KUKA KRL program: MyProgram_012().src

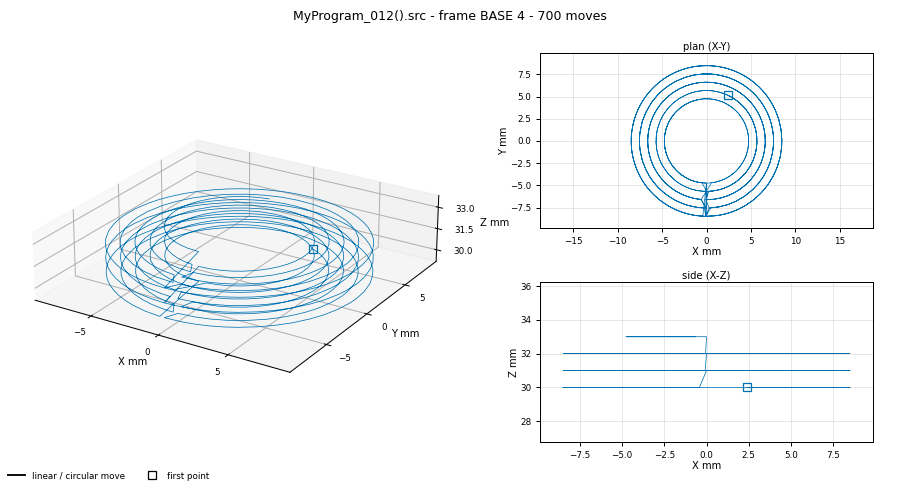
[picture p0: tool path of MyProgram_012().src in frame BASE 4, 700 of 700 moves have a stored position in this frame; points joined in program order, loops and branches not executed]
&ACCESS RVP
&REL 1
&PARAM TEMPLATE = C:\KRC\Roboter\Template\vorgabe
&PARAM EDITMASK = *
DEF MyProgram_012()
; ---- Setting reference (Base) ----
$BASE = BASE_DATA[4]

; --------------------------
; ---- Setting tool (TCP) ----
$TOOL = TOOL_DATA[3]
; --------------------------

$VEL.CP = VEL_APROX_PRINT
Startdeposition()
$VEL.CP = VEL_PRINT
LIN {X 2.4123,Y 5.1442,Z 30,A -2.4126,B 0,C 0,E1 0.1598,E2 90.0723} C_DIS
LIN {X 3.1461,Y 4.7312,Z 30,A -2.403,B 0,C 0,E1 0.1598,E2 90.0723} C_DIS
LIN {X 3.8114,Y 4.215,Z 30,A -2.4004,B 0,C 0,E1 0.1598,E2 90.0723} C_DIS
LIN {X 4.392,Y 3.6051,Z 30,A -2.4048,B 0,C 0,E1 0.1598,E2 90.0721} C_DIS
LIN {X 4.8767,Y 2.9165,Z 30,A -2.4161,B 0,C 0,E1 0.1598,E2 90.0721} C_DIS
LIN {X 5.2536,Y 2.1636,Z 30,A -2.4342,B 0,C 0,E1 0.1598,E2 90.072} C_DIS
LIN {X 5.5158,Y 1.3634,Z 30,A -2.4585,B 0,C 0,E1 0.1598,E2 90.072} C_DIS
LIN {X 5.6573,Y 0.5334,Z 30,A -2.4886,B 0,C 0,E1 0.1598,E2 90.0719} C_DIS
LIN {X 5.6741,Y -0.3085,Z 30,A -2.5238,B 0,C 0,E1 0.1598,E2 90.0719} C_DIS
LIN {X 5.567,Y -1.1438,Z 30,A -2.5633,B 0,C 0,E1 0.1598,E2 90.0718} C_DIS
LIN {X 5.3364,Y -1.9538,Z 30,A -2.6062,B 0,C 0,E1 0.1598,E2 90.0718} C_DIS
LIN {X 4.9891,Y -2.721,Z 30,A -2.6517,B 0,C 0,E1 0.1598,E2 90.0718} C_DIS
LIN {X 4.5312,Y -3.4277,Z 30,A -2.6986,B 0,C 0,E1 0.1598,E2 90.0718} C_DIS
LIN {X 3.9758,Y -4.0606,Z 30,A -2.746,B 0,C 0,E1 0.1598,E2 90.0718} C_DIS
LIN {X 3.3312,Y -4.6025,Z 30,A -2.7928,B 0,C 0,E1 0.1598,E2 90.0718} C_DIS
LIN {X 2.6147,Y -5.0448,Z 30,A -2.8379,B 0,C 0,E1 0.1598,E2 90.0717} C_DIS
LIN {X 1.8405,Y -5.3759,Z 30,A -2.8805,B 0,C 0,E1 0.1598,E2 90.0717} C_DIS
LIN {X 1.0258,Y -5.5886,Z 30,A -2.9194,B 0,C 0,E1 0.1598,E2 90.0717} C_DIS
LIN {X 0.1887,Y -5.6795,Z 30,A -2.954,B 0,C 0,E1 0.1598,E2 90.0717} C_DIS
LIN {X 0.1887,Y -5.6795,Z 30,A -2.954,B 0,C 0,E1 0.1598,E2 90.0717} C_DIS
Enddeposition()
LIN {X -0.0561,Y -6.623,Z 30,A -3.0021,B 0,C 0,E1 0.1598,E2 90.0704} C_DIS
Startdeposition()
$VEL.CP = VEL_PRINT
LIN {X 0.9035,Y -6.5557,Z 30,A -2.9651,B 0,C 0,E1 0.1598,E2 90.0716} C_DIS
LIN {X 1.6588,Y -6.4076,Z 30,A -2.9312,B 0,C 0,E1 0.1598,E2 90.0716} C_DIS
LIN {X 2.3917,Y -6.1725,Z 30,A -2.8943,B 0,C 0,E1 0.1598,E2 90.0716} C_DIS
LIN {X 3.0924,Y -5.8533,Z 30,A -2.855,B 0,C 0,E1 0.1598,E2 90.0717} C_DIS
LIN {X 3.7497,Y -5.4527,Z 30,A -2.8138,B 0,C 0,E1 0.1598,E2 90.0717} C_DIS
LIN {X 4.3594,Y -4.983,Z 30,A -2.7714,B 0,C 0,E1 0.1598,E2 90.0717} C_DIS
LIN {X 4.9078,Y -4.4428,Z 30,A -2.7282,B 0,C 0,E1 0.1598,E2 90.0717} C_DIS
LIN {X 5.3882,Y -3.8416,Z 30,A -2.6849,B 0,C 0,E1 0.1598,E2 90.0718} C_DIS
LIN {X 5.7983,Y -3.1903,Z 30,A -2.6421,B 0,C 0,E1 0.1598,E2 90.0718} C_DIS
LIN {X 6.1306,Y -2.4959,Z 30,A -2.6003,B 0,C 0,E1 0.1598,E2 90.0718} C_DIS
LIN {X 6.3796,Y -1.7675,Z 30,A -2.5601,B 0,C 0,E1 0.1598,E2 90.0718} C_DIS
LIN {X 6.5402,Y -1.0147,Z 30,A -2.5221,B 0,C 0,E1 0.1598,E2 90.0718} C_DIS
LIN {X 6.613,Y -0.2485,Z 30,A -2.4868,B 0,C 0,E1 0.1598,E2 90.0719} C_DIS
LIN {X 6.5976,Y 0.5209,Z 30,A -2.4546,B 0,C 0,E1 0.1598,E2 90.0719} C_DIS
LIN {X 6.4945,Y 1.2838,Z 30,A -2.4259,B 0,C 0,E1 0.1598,E2 90.072} C_DIS
LIN {X 6.2995,Y 2.0284,Z 30,A -2.4014,B 0,C 0,E1 0.1598,E2 90.072} C_DIS
LIN {X 6.0209,Y 2.7458,Z 30,A -2.3812,B 0,C 0,E1 0.1598,E2 90.072} C_DIS
LIN {X 5.6618,Y 3.4265,Z 30,A -2.3655,B 0,C 0,E1 0.1598,E2 90.0721} C_DIS
LIN {X 5.2259,Y 4.0609,Z 30,A -2.3547,B 0,C 0,E1 0.1598,E2 90.0721} C_DIS
LIN {X 4.7191,Y 4.6402,Z 30,A -2.3488,B 0,C 0,E1 0.1598,E2 90.0722} C_DIS
LIN {X 4.1479,Y 5.156,Z 30,A -2.348,B 0,C 0,E1 0.1598,E2 90.0722} C_DIS
LIN {X 3.5214,Y 5.6029,Z 30,A -2.3521,B 0,C 0,E1 0.1598,E2 90.0723} C_DIS
LIN {X 2.8468,Y 5.9734,Z 30,A -2.3613,B 0,C 0,E1 0.1598,E2 90.0723} C_DIS
LIN {X 2.1347,Y 6.2654,Z 30,A -2.3753,B 0,C 0,E1 0.1598,E2 90.0723} C_DIS
LIN {X 1.393,Y 6.4721,Z 30,A -2.3939,B 0,C 0,E1 0.1598,E2 90.0723} C_DIS
LIN {X 0.6321,Y 6.5887,Z 30,A -2.417,B 0,C 0,E1 0.1598,E2 90.0723} C_DIS
LIN {X -0.137,Y 6.616,Z 30,A -2.4443,B 0,C 0,E1 0.1598,E2 90.0723} C_DIS
LIN {X -0.9042,Y 6.5562,Z 30,A -2.4751,B 0,C 0,E1 0.1598,E2 90.0723} C_DIS
LIN {X -1.6593,Y 6.4071,Z 30,A -2.5093,B 0,C 0,E1 0.1598,E2 90.0723} C_DIS
LIN {X -2.3924,Y 6.1721,Z 30,A -2.5462,B 0,C 0,E1 0.1598,E2 90.0722} C_DIS
LIN {X -3.093,Y 5.8529,Z 30,A -2.5855,B 0,C 0,E1 0.1598,E2 90.0721} C_DIS
LIN {X -3.7524,Y 5.4556,Z 30,A -2.6266,B 0,C 0,E1 0.1598,E2 90.072} C_DIS
LIN {X -4.3593,Y 4.9822,Z 30,A -2.669,B 0,C 0,E1 0.1598,E2 90.072} C_DIS
LIN {X -4.9079,Y 4.4421,Z 30,A -2.712,B 0,C 0,E1 0.1598,E2 90.0718} C_DIS
LIN {X -5.3904,Y 3.8421,Z 30,A -2.7551,B 0,C 0,E1 0.1598,E2 90.0718} C_DIS
LIN {X -5.8017,Y 3.1913,Z 30,A -2.7977,B 0,C 0,E1 0.1598,E2 90.0716} C_DIS
LIN {X -6.132,Y 2.496,Z 30,A -2.8392,B 0,C 0,E1 0.1598,E2 90.0716} C_DIS
LIN {X -6.3803,Y 1.7674,Z 30,A -2.8791,B 0,C 0,E1 0.1598,E2 90.0715} C_DIS
LIN {X -6.5428,Y 1.015,Z 30,A -2.9168,B 0,C 0,E1 0.1598,E2 90.0714} C_DIS
LIN {X -6.6157,Y 0.2486,Z 30,A -2.9518,B 0,C 0,E1 0.1598,E2 90.0714} C_DIS
LIN {X -6.5995,Y -0.521,Z 30,A -2.9837,B 0,C 0,E1 0.1598,E2 90.0713} C_DIS
LIN {X -6.493,Y -1.2834,Z 30,A -3.0121,B 0,C 0,E1 0.1598,E2 90.0713} C_DIS
LIN {X -6.2988,Y -2.0281,Z 30,A -3.0364,B 0,C 0,E1 0.1598,E2 90.0713} C_DIS
LIN {X -6.0221,Y -2.7462,Z 30,A -3.0566,B 0,C 0,E1 0.1598,E2 90.0713} C_DIS
LIN {X -5.6621,Y -3.4265,Z 30,A -3.0722,B 0,C 0,E1 0.1598,E2 90.0713} C_DIS
LIN {X -5.2258,Y -4.0606,Z 30,A -3.083,B 0,C 0,E1 0.1598,E2 90.0713} C_DIS
LIN {X -4.7193,Y -4.6402,Z 30,A -3.089,B 0,C 0,E1 0.1598,E2 90.0713} C_DIS
LIN {X -4.1488,Y -5.157,Z 30,A -3.09,B 0,C 0,E1 0.1598,E2 90.0713} C_DIS
LIN {X -3.5234,Y -5.6058,Z 30,A -3.0861,B 0,C 0,E1 0.1598,E2 90.0713} C_DIS
LIN {X -2.8478,Y -5.9745,Z 30,A -3.077,B 0,C 0,E1 0.1598,E2 90.0713} C_DIS
LIN {X -2.1347,Y -6.2644,Z 30,A -3.0631,B 0,C 0,E1 0.1598,E2 90.0714} C_DIS
LIN {X -1.3938,Y -6.4732,Z 30,A -3.0448,B 0,C 0,E1 0.1598,E2 90.0714} C_DIS
LIN {X -0.6329,Y -6.5897,Z 30,A -3.0219,B 0,C 0,E1 0.1598,E2 90.0715} C_DIS
LIN {X -0.6329,Y -6.5897,Z 30,A -3.0219,B 0,C 0,E1 0.1598,E2 90.0715} C_DIS
Enddeposition()
LIN {X -0.0547,Y -7.5529,Z 30,A -3.0406,B 0,C 0,E1 0.1598,E2 90.0703} C_DIS
Startdeposition()
$VEL.CP = VEL_PRINT
LIN {X -0.7724,Y -7.5177,Z 30,A -3.0665,B 0,C 0,E1 0.1598,E2 90.0714} C_DIS
LIN {X -1.851,Y -7.322,Z 30,A -3.0978,B 0,C 0,E1 0.1598,E2 90.0714} C_DIS
LIN {X -2.6875,Y -7.0585,Z 30,A -3.1173,B 0,C 0,E1 0.1598,E2 90.0714} C_DIS
LIN {X -3.4877,Y -6.6995,Z 30,A -3.1314,B 0,C 0,E1 0.1598,E2 90.0714} C_DIS
LIN {X -4.5316,Y -6.0476,Z 30,A -3.1419,B 0,C 0,E1 0.1598,E2 90.0712} C_DIS
LIN {X -5.2966,Y -5.385,Z 30,A -3.1419,B 0,C 0,E1 0.1598,E2 90.0712} C_DIS
LIN {X -5.8428,Y -4.7872,Z 30,A -3.1367,B 0,C 0,E1 0.1598,E2 90.0712} C_DIS
LIN {X -6.3205,Y -4.1335,Z 30,A -3.1265,B 0,C 0,E1 0.1598,E2 90.0712} C_DIS
LIN {X -6.8204,Y -3.2535,Z 30,A -3.1074,B 0,C 0,E1 0.1598,E2 90.0709} C_DIS
LIN {X -7.2077,Y -2.2699,Z 30,A -3.08,B 0,C 0,E1 0.1598,E2 90.0709} C_DIS
LIN {X -7.497,Y -0.9548,Z 30,A -3.0348,B 0,C 0,E1 0.1598,E2 90.0707} C_DIS
LIN {X -7.5586,Y 0,Z 30,A -2.997,B 0,C 0,E1 0.1598,E2 90.071} C_DIS
LIN {X -7.4963,Y 0.9605,Z 30,A -2.9542,B 0,C 0,E1 0.1598,E2 90.0712} C_DIS
LIN {X -7.2248,Y 2.2151,Z 30,A -2.8909,B 0,C 0,E1 0.1598,E2 90.0709} C_DIS
LIN {X -6.777,Y 3.3346,Z 30,A -2.8272,B 0,C 0,E1 0.1598,E2 90.0711} C_DIS
LIN {X -6.1243,Y 4.4288,Z 30,A -2.7571,B 0,C 0,E1 0.1598,E2 90.0713} C_DIS
LIN {X -5.5112,Y 5.165,Z 30,A -2.7037,B 0,C 0,E1 0.1598,E2 90.0717} C_DIS
LIN {X -4.9608,Y 5.6982,Z 30,A -2.661,B 0,C 0,E1 0.1598,E2 90.0719} C_DIS
LIN {X -4.3575,Y 6.171,Z 30,A -2.6188,B 0,C 0,E1 0.1598,E2 90.0719} C_DIS
LIN {X -3.5431,Y 6.6752,Z 30,A -2.5675,B 0,C 0,E1 0.1598,E2 90.072} C_DIS
LIN {X -2.4286,Y 7.1518,Z 30,A -2.5062,B 0,C 0,E1 0.1598,E2 90.0721} C_DIS
LIN {X -1.5729,Y 7.3873,Z 30,A -2.4648,B 0,C 0,E1 0.1598,E2 90.0723} C_DIS
LIN {X -0.3721,Y 7.549,Z 30,A -2.4136,B 0,C 0,E1 0.1598,E2 90.0723} C_DIS
LIN {X 0.6118,Y 7.5328,Z 30,A -2.378,B 0,C 0,E1 0.1598,E2 90.0723} C_DIS
LIN {X 1.7598,Y 7.3459,Z 30,A -2.3435,B 0,C 0,E1 0.1598,E2 90.0724} C_DIS
LIN {X 2.486,Y 7.1371,Z 30,A -2.3255,B 0,C 0,E1 0.1598,E2 90.0724} C_DIS
LIN {X 3.3884,Y 6.7498,Z 30,A -2.3086,B 0,C 0,E1 0.1598,E2 90.0724} C_DIS
LIN {X 4.071,Y 6.3612,Z 30,A -2.2999,B 0,C 0,E1 0.1598,E2 90.0724} C_DIS
LIN {X 4.7103,Y 5.9047,Z 30,A -2.2957,B 0,C 0,E1 0.1598,E2 90.0724} C_DIS
LIN {X 5.2981,Y 5.3837,Z 30,A -2.2961,B 0,C 0,E1 0.1598,E2 90.0724} C_DIS
LIN {X 5.8284,Y 4.8041,Z 30,A -2.3011,B 0,C 0,E1 0.1598,E2 90.0723} C_DIS
LIN {X 6.2957,Y 4.1726,Z 30,A -2.3107,B 0,C 0,E1 0.1598,E2 90.0723} C_DIS
LIN {X 6.6959,Y 3.4965,Z 30,A -2.3247,B 0,C 0,E1 0.1598,E2 90.0722} C_DIS
LIN {X 7.0228,Y 2.7821,Z 30,A -2.343,B 0,C 0,E1 0.1598,E2 90.0722} C_DIS
LIN {X 7.3273,Y 1.8485,Z 30,A -2.3712,B 0,C 0,E1 0.1598,E2 90.0718} C_DIS
LIN {X 7.5275,Y 0.6253,Z 30,A -2.4155,B 0,C 0,E1 0.1598,E2 90.0714} C_DIS
LIN {X 7.556,Y -0.1257,Z 30,A -2.4469,B 0,C 0,E1 0.1598,E2 90.0718} C_DIS
LIN {X 7.4453,Y -1.2667,Z 30,A -2.4994,B 0,C 0,E1 0.1598,E2 90.0716} C_DIS
LIN {X 7.1403,Y -2.4763,Z 30,A -2.5621,B 0,C 0,E1 0.1598,E2 90.0714} C_DIS
LIN {X 6.7973,Y -3.3011,Z 30,A -2.6101,B 0,C 0,E1 0.1598,E2 90.0716} C_DIS
LIN {X 6.3336,Y -4.1158,Z 30,A -2.6619,B 0,C 0,E1 0.1598,E2 90.0716} C_DIS
LIN {X 5.8945,Y -4.7239,Z 30,A -2.7041,B 0,C 0,E1 0.1598,E2 90.0718} C_DIS
LIN {X 5.2662,Y -5.4196,Z 30,A -2.7567,B 0,C 0,E1 0.1598,E2 90.0716} C_DIS
LIN {X 4.2992,Y -6.2142,Z 30,A -2.826,B 0,C 0,E1 0.1598,E2 90.0716} C_DIS
LIN {X 3.3206,Y -6.7878,Z 30,A -2.8864,B 0,C 0,E1 0.1598,E2 90.0716} C_DIS
LIN {X 2.3699,Y -7.1764,Z 30,A -2.9379,B 0,C 0,E1 0.1598,E2 90.0716} C_DIS
LIN {X 1.4049,Y -7.4218,Z 30,A -2.9838,B 0,C 0,E1 0.1598,E2 90.0716} C_DIS
LIN {X 0.2911,Y -7.5523,Z 30,A -3.0302,B 0,C 0,E1 0.1598,E2 90.0716} C_DIS
LIN {X 0.2911,Y -7.5523,Z 30,A -3.0302,B 0,C 0,E1 0.1598,E2 90.0716} C_DIS
Enddeposition()
LIN {X -0.0783,Y -8.4901,Z 30,A -3.0826,B 0,C 0,E1 0.1598,E2 90.0703} C_DIS
Startdeposition()
$VEL.CP = VEL_PRINT
LIN {X 1.2283,Y -8.3988,Z 30,A -3.0319,B 0,C 0,E1 0.1598,E2 90.0715} C_DIS
LIN {X 2.0607,Y -8.2346,Z 30,A -2.9945,B 0,C 0,E1 0.1598,E2 90.0715} C_DIS
LIN {X 2.8724,Y -7.9881,Z 30,A -2.9542,B 0,C 0,E1 0.1598,E2 90.0716} C_DIS
LIN {X 3.6554,Y -7.6615,Z 30,A -2.9116,B 0,C 0,E1 0.1598,E2 90.0716} C_DIS
LIN {X 4.4018,Y -7.2582,Z 30,A -2.867,B 0,C 0,E1 0.1598,E2 90.0716} C_DIS
LIN {X 5.4213,Y -6.535,Z 30,A -2.7987,B 0,C 0,E1 0.1598,E2 90.0716} C_DIS
LIN {X 6.1607,Y -5.8374,Z 30,A -2.7419,B 0,C 0,E1 0.1598,E2 90.0716} C_DIS
LIN {X 6.8736,Y -4.9869,Z 30,A -2.6793,B 0,C 0,E1 0.1598,E2 90.0716} C_DIS
LIN {X 7.4968,Y -3.9772,Z 30,A -2.6132,B 0,C 0,E1 0.1598,E2 90.0716} C_DIS
LIN {X 7.9383,Y -3.0124,Z 30,A -2.5558,B 0,C 0,E1 0.1598,E2 90.0716} C_DIS
LIN {X 8.2832,Y -1.8682,Z 30,A -2.4943,B 0,C 0,E1 0.1598,E2 90.0716} C_DIS
LIN {X 8.4617,Y -0.6618,Z 30,A -2.4361,B 0,C 0,E1 0.1598,E2 90.0714} C_DIS
LIN {X 8.4909,Y 0.0804,Z 30,A -2.4038,B 0,C 0,E1 0.1598,E2 90.0719} C_DIS
LIN {X 8.399,Y 1.224,Z 30,A -2.3581,B 0,C 0,E1 0.1598,E2 90.0716} C_DIS
LIN {X 8.1382,Y 2.4222,Z 30,A -2.3167,B 0,C 0,E1 0.1598,E2 90.0716} C_DIS
LIN {X 7.7294,Y 3.5063,Z 30,A -2.2856,B 0,C 0,E1 0.1598,E2 90.0718} C_DIS
LIN {X 7.234,Y 4.4442,Z 30,A -2.2641,B 0,C 0,E1 0.1598,E2 90.0719} C_DIS
LIN {X 6.6525,Y 5.2763,Z 30,A -2.2503,B 0,C 0,E1 0.1598,E2 90.0721} C_DIS
LIN {X 5.9407,Y 6.0622,Z 30,A -2.2433,B 0,C 0,E1 0.1598,E2 90.0722} C_DIS
LIN {X 5.3057,Y 6.6248,Z 30,A -2.2429,B 0,C 0,E1 0.1598,E2 90.0724} C_DIS
LIN {X 4.6179,Y 7.1212,Z 30,A -2.2473,B 0,C 0,E1 0.1598,E2 90.0724} C_DIS
LIN {X 3.8839,Y 7.5467,Z 30,A -2.2564,B 0,C 0,E1 0.1598,E2 90.0724} C_DIS
LIN {X 3.1112,Y 7.8967,Z 30,A -2.2701,B 0,C 0,E1 0.1598,E2 90.0724} C_DIS
LIN {X 2.3074,Y 8.168,Z 30,A -2.2883,B 0,C 0,E1 0.1598,E2 90.0724} C_DIS
LIN {X 1.2716,Y 8.395,Z 30,A -2.3169,B 0,C 0,E1 0.1598,E2 90.0724} C_DIS
LIN {X -0.0129,Y 8.4922,Z 30,A -2.3603,B 0,C 0,E1 0.1598,E2 90.0724} C_DIS
LIN {X -1.2348,Y 8.3979,Z 30,A -2.4094,B 0,C 0,E1 0.1598,E2 90.0724} C_DIS
LIN {X -2.0651,Y 8.2336,Z 30,A -2.447,B 0,C 0,E1 0.1598,E2 90.0723} C_DIS
LIN {X -2.8747,Y 7.9871,Z 30,A -2.4873,B 0,C 0,E1 0.1598,E2 90.0723} C_DIS
LIN {X -3.6558,Y 7.6613,Z 30,A -2.5299,B 0,C 0,E1 0.1598,E2 90.0721} C_DIS
LIN {X -4.4004,Y 7.2589,Z 30,A -2.5743,B 0,C 0,E1 0.1598,E2 90.0721} C_DIS
LIN {X -5.1011,Y 6.7843,Z 30,A -2.6202,B 0,C 0,E1 0.1598,E2 90.072} C_DIS
LIN {X -5.751,Y 6.2423,Z 30,A -2.667,B 0,C 0,E1 0.1598,E2 90.0719} C_DIS
LIN {X -6.3439,Y 5.6383,Z 30,A -2.7143,B 0,C 0,E1 0.1598,E2 90.0718} C_DIS
LIN {X -6.8734,Y 4.9781,Z 30,A -2.7617,B 0,C 0,E1 0.1598,E2 90.0717} C_DIS
LIN {X -7.3356,Y 4.2691,Z 30,A -2.8086,B 0,C 0,E1 0.1598,E2 90.0716} C_DIS
LIN {X -7.7243,Y 3.5173,Z 30,A -2.8546,B 0,C 0,E1 0.1598,E2 90.0715} C_DIS
LIN {X -8.1292,Y 2.4512,Z 30,A -2.9142,B 0,C 0,E1 0.1598,E2 90.0712} C_DIS
LIN {X -8.4129,Y 1.1577,Z 30,A -2.9789,B 0,C 0,E1 0.1598,E2 90.0708} C_DIS
LIN {X -8.4915,Y 0.0524,Z 30,A -3.0287,B 0,C 0,E1 0.1598,E2 90.0709} C_DIS
LIN {X -8.4293,Y -1.0187,Z 30,A -3.0716,B 0,C 0,E1 0.1598,E2 90.0709} C_DIS
LIN {X -8.2649,Y -1.9515,Z 30,A -3.105,B 0,C 0,E1 0.1598,E2 90.0709} C_DIS
LIN {X -7.956,Y -2.9554,Z 30,A -3.1361,B 0,C 0,E1 0.1598,E2 90.0709} C_DIS
LIN {X -7.6249,Y -3.7276,Z 30,A -3.1567,B 0,C 0,E1 0.1598,E2 90.071} C_DIS
LIN {X -7.2188,Y -4.4632,Z 30,A -3.173,B 0,C 0,E1 0.1598,E2 90.071} C_DIS
LIN {X -6.7419,Y -5.1551,Z 30,A -3.1847,B 0,C 0,E1 0.1598,E2 90.071} C_DIS
LIN {X -6.1988,Y -5.7963,Z 30,A -3.192,B 0,C 0,E1 0.1598,E2 90.071} C_DIS
LIN {X -5.5951,Y -6.3808,Z 30,A -3.1946,B 0,C 0,E1 0.1598,E2 90.0711} C_DIS
LIN {X -4.9367,Y -6.9029,Z 30,A -3.1926,B 0,C 0,E1 0.1598,E2 90.0711} C_DIS
LIN {X -4.2298,Y -7.3574,Z 30,A -3.186,B 0,C 0,E1 0.1598,E2 90.0712} C_DIS
LIN {X -3.4817,Y -7.7402,Z 30,A -3.1748,B 0,C 0,E1 0.1598,E2 90.0712} C_DIS
LIN {X -2.6992,Y -8.0469,Z 30,A -3.1592,B 0,C 0,E1 0.1598,E2 90.0713} C_DIS
LIN {X -1.5972,Y -8.3401,Z 30,A -3.1312,B 0,C 0,E1 0.1598,E2 90.0713} C_DIS
LIN {X -0.4191,Y -8.4815,Z 30,A -3.0941,B 0,C 0,E1 0.1598,E2 90.0714} C_DIS
LIN {X -0.4191,Y -8.4815,Z 30,A -3.0941,B 0,C 0,E1 0.1598,E2 90.0714} C_DIS
Enddeposition()
LIN {X 0.0007,Y -4.7567,Z 31,A -2.9056,B 0,C 0,E1 0.1598,E2 90.0604} C_DIS
Startdeposition()
$VEL.CP = VEL_PRINT
LIN {X 0.0007,Y -4.7567,Z 31,A -2.9113,B 0,C 0,E1 0.1598,E2 90.0661} C_DIS
LIN {X -0.9854,Y -4.646,Z 31,A -2.9477,B 0,C 0,E1 0.1598,E2 90.071} C_DIS
LIN {X -1.5934,Y -4.4747,Z 31,A -2.9634,B 0,C 0,E1 0.1598,E2 90.0716} C_DIS
LIN {X -2.2528,Y -4.1814,Z 31,A -2.9751,B 0,C 0,E1 0.1598,E2 90.0716} C_DIS
LIN {X -2.8616,Y -3.7934,Z 31,A -2.981,B 0,C 0,E1 0.1598,E2 90.0716} C_DIS
LIN {X -3.4035,Y -3.3161,Z 31,A -2.9806,B 0,C 0,E1 0.1598,E2 90.0715} C_DIS
LIN {X -3.8656,Y -2.7613,Z 31,A -2.9741,B 0,C 0,E1 0.1598,E2 90.0715} C_DIS
LIN {X -4.2384,Y -2.1432,Z 31,A -2.9615,B 0,C 0,E1 0.1598,E2 90.0715} C_DIS
LIN {X -4.5137,Y -1.4761,Z 31,A -2.9434,B 0,C 0,E1 0.1598,E2 90.0715} C_DIS
LIN {X -4.6862,Y -0.7754,Z 31,A -2.9201,B 0,C 0,E1 0.1598,E2 90.0715} C_DIS
LIN {X -4.7489,Y 0.0339,Z 31,A -2.8881,B 0,C 0,E1 0.1598,E2 90.0714} C_DIS
LIN {X -4.7052,Y 0.6641,Z 31,A -2.8599,B 0,C 0,E1 0.1598,E2 90.0716} C_DIS
LIN {X -4.5493,Y 1.3691,Z 31,A -2.8243,B 0,C 0,E1 0.1598,E2 90.0716} C_DIS
LIN {X -4.288,Y 2.0419,Z 31,A -2.7863,B 0,C 0,E1 0.1598,E2 90.0716} C_DIS
LIN {X -3.9291,Y 2.6681,Z 31,A -2.7466,B 0,C 0,E1 0.1598,E2 90.0717} C_DIS
LIN {X -3.4173,Y 3.2982,Z 31,A -2.7011,B 0,C 0,E1 0.1598,E2 90.0717} C_DIS
LIN {X -2.9495,Y 3.7225,Z 31,A -2.666,B 0,C 0,E1 0.1598,E2 90.0719} C_DIS
LIN {X -2.351,Y 4.1257,Z 31,A -2.6269,B 0,C 0,E1 0.1598,E2 90.0719} C_DIS
LIN {X -1.6993,Y 4.4357,Z 31,A -2.5898,B 0,C 0,E1 0.1598,E2 90.0721} C_DIS
LIN {X -1.0077,Y 4.6421,Z 31,A -2.5556,B 0,C 0,E1 0.1598,E2 90.0721} C_DIS
LIN {X -0.2929,Y 4.743,Z 31,A -2.525,B 0,C 0,E1 0.1598,E2 90.0722} C_DIS
LIN {X 0.429,Y 4.7318,Z 31,A -2.4988,B 0,C 0,E1 0.1598,E2 90.0722} C_DIS
LIN {X 1.1413,Y 4.6134,Z 31,A -2.4776,B 0,C 0,E1 0.1598,E2 90.0722} C_DIS
LIN {X 1.8264,Y 4.3854,Z 31,A -2.462,B 0,C 0,E1 0.1598,E2 90.0722} C_DIS
LIN {X 2.4694,Y 4.0573,Z 31,A -2.4522,B 0,C 0,E1 0.1598,E2 90.0722} C_DIS
LIN {X 3.055,Y 3.6355,Z 31,A -2.4484,B 0,C 0,E1 0.1598,E2 90.0722} C_DIS
LIN {X 3.571,Y 3.1311,Z 31,A -2.4508,B 0,C 0,E1 0.1598,E2 90.0722} C_DIS
LIN {X 4.0522,Y 2.4774,Z 31,A -2.4607,B 0,C 0,E1 0.1598,E2 90.072} C_DIS
LIN {X 4.3468,Y 1.9185,Z 31,A -2.4737,B 0,C 0,E1 0.1598,E2 90.072} C_DIS
LIN {X 4.5876,Y 1.2378,Z 31,A -2.4937,B 0,C 0,E1 0.1598,E2 90.072} C_DIS
LIN {X 4.7223,Y 0.5286,Z 31,A -2.5189,B 0,C 0,E1 0.1598,E2 90.072} C_DIS
LIN {X 4.7478,Y -0.1929,Z 31,A -2.5486,B 0,C 0,E1 0.1598,E2 90.0719} C_DIS
LIN {X 4.6622,Y -0.9096,Z 31,A -2.5822,B 0,C 0,E1 0.1598,E2 90.0719} C_DIS
LIN {X 4.4711,Y -1.6058,Z 31,A -2.6189,B 0,C 0,E1 0.1598,E2 90.0719} C_DIS
LIN {X 4.1763,Y -2.2647,Z 31,A -2.6578,B 0,C 0,E1 0.1598,E2 90.0718} C_DIS
LIN {X 3.6774,Y -3.0169,Z 31,A -2.708,B 0,C 0,E1 0.1598,E2 90.0716} C_DIS
LIN {X 3.187,Y -3.5251,Z 31,A -2.7478,B 0,C 0,E1 0.1598,E2 90.0718} C_DIS
LIN {X 2.6039,Y -3.9716,Z 31,A -2.7883,B 0,C 0,E1 0.1598,E2 90.0718} C_DIS
LIN {X 1.9608,Y -4.3257,Z 31,A -2.827,B 0,C 0,E1 0.1598,E2 90.0718} C_DIS
LIN {X 1.271,Y -4.5773,Z 31,A -2.863,B 0,C 0,E1 0.1598,E2 90.0718} C_DIS
LIN {X 0.5507,Y -4.7196,Z 31,A -2.8955,B 0,C 0,E1 0.1598,E2 90.0718} C_DIS
LIN {X 0.5507,Y -4.7196,Z 31,A -2.8955,B 0,C 0,E1 0.1598,E2 90.0718} C_DIS
Enddeposition()
LIN {X -0.0222,Y -5.6862,Z 31,A -2.9566,B 0,C 0,E1 0.1598,E2 90.0705} C_DIS
Startdeposition()
$VEL.CP = VEL_PRINT
LIN {X 0.6087,Y -5.65,Z 31,A -2.933,B 0,C 0,E1 0.1598,E2 90.0716} C_DIS
LIN {X 1.4368,Y -5.4973,Z 31,A -2.8962,B 0,C 0,E1 0.1598,E2 90.0717} C_DIS
LIN {X 2.2335,Y -5.2251,Z 31,A -2.8553,B 0,C 0,E1 0.1598,E2 90.0717} C_DIS
LIN {X 2.9807,Y -4.837,Z 31,A -2.8114,B 0,C 0,E1 0.1598,E2 90.0717} C_DIS
LIN {X 3.663,Y -4.3436,Z 31,A -2.7653,B 0,C 0,E1 0.1598,E2 90.0717} C_DIS
LIN {X 4.265,Y -3.7549,Z 31,A -2.7181,B 0,C 0,E1 0.1598,E2 90.0717} C_DIS
LIN {X 4.7728,Y -3.0833,Z 31,A -2.6708,B 0,C 0,E1 0.1598,E2 90.0717} C_DIS
LIN {X 5.1767,Y -2.3445,Z 31,A -2.6244,B 0,C 0,E1 0.1598,E2 90.0717} C_DIS
LIN {X 5.4664,Y -1.5538,Z 31,A -2.5801,B 0,C 0,E1 0.1598,E2 90.0717} C_DIS
LIN {X 5.6359,Y -0.7289,Z 31,A -2.5387,B 0,C 0,E1 0.1598,E2 90.0718} C_DIS
LIN {X 5.6819,Y 0.1119,Z 31,A -2.5012,B 0,C 0,E1 0.1598,E2 90.0718} C_DIS
LIN {X 5.6017,Y 0.9501,Z 31,A -2.4685,B 0,C 0,E1 0.1598,E2 90.0718} C_DIS
LIN {X 5.3999,Y 1.7675,Z 31,A -2.4412,B 0,C 0,E1 0.1598,E2 90.0719} C_DIS
LIN {X 5.0795,Y 2.5461,Z 31,A -2.4199,B 0,C 0,E1 0.1598,E2 90.0719} C_DIS
LIN {X 4.6477,Y 3.2688,Z 31,A -2.4051,B 0,C 0,E1 0.1598,E2 90.0721} C_DIS
LIN {X 4.1141,Y 3.9203,Z 31,A -2.3971,B 0,C 0,E1 0.1598,E2 90.0721} C_DIS
LIN {X 3.4893,Y 4.4847,Z 31,A -2.3963,B 0,C 0,E1 0.1598,E2 90.0721} C_DIS
LIN {X 2.788,Y 4.9507,Z 31,A -2.4024,B 0,C 0,E1 0.1598,E2 90.0722} C_DIS
LIN {X 2.0258,Y 5.3083,Z 31,A -2.4154,B 0,C 0,E1 0.1598,E2 90.0722} C_DIS
LIN {X 1.2194,Y 5.5501,Z 31,A -2.4349,B 0,C 0,E1 0.1598,E2 90.0722} C_DIS
LIN {X 0.3859,Y 5.6706,Z 31,A -2.4606,B 0,C 0,E1 0.1598,E2 90.0722} C_DIS
LIN {X -0.4562,Y 5.6648,Z 31,A -2.4919,B 0,C 0,E1 0.1598,E2 90.0722} C_DIS
LIN {X -1.2889,Y 5.5376,Z 31,A -2.528,B 0,C 0,E1 0.1598,E2 90.0722} C_DIS
LIN {X -2.0946,Y 5.2914,Z 31,A -2.5681,B 0,C 0,E1 0.1598,E2 90.0722} C_DIS
LIN {X -3.1653,Y 4.7215,Z 31,A -2.6315,B 0,C 0,E1 0.1598,E2 90.0719} C_DIS
LIN {X -3.7946,Y 4.2342,Z 31,A -2.6754,B 0,C 0,E1 0.1598,E2 90.0719} C_DIS
LIN {X -4.3482,Y 3.6623,Z 31,A -2.7199,B 0,C 0,E1 0.1598,E2 90.0718} C_DIS
LIN {X -4.8163,Y 3.0187,Z 31,A -2.7643,B 0,C 0,E1 0.1598,E2 90.0717} C_DIS
LIN {X -5.1907,Y 2.3165,Z 31,A -2.8077,B 0,C 0,E1 0.1598,E2 90.0716} C_DIS
LIN {X -5.5459,Y 1.2725,Z 31,A -2.8647,B 0,C 0,E1 0.1598,E2 90.0712} C_DIS
LIN {X -5.6708,Y 0.411,Z 31,A -2.9058,B 0,C 0,E1 0.1598,E2 90.0713} C_DIS
LIN {X -5.6783,Y -0.2853,Z 31,A -2.9356,B 0,C 0,E1 0.1598,E2 90.0713} C_DIS
LIN {X -5.6004,Y -0.9773,Z 31,A -2.962,B 0,C 0,E1 0.1598,E2 90.0713} C_DIS
LIN {X -5.4408,Y -1.6552,Z 31,A -2.9849,B 0,C 0,E1 0.1598,E2 90.0713} C_DIS
LIN {X -5.1966,Y -2.3074,Z 31,A -3.0035,B 0,C 0,E1 0.1598,E2 90.0713} C_DIS
LIN {X -4.8739,Y -2.9245,Z 31,A -3.0178,B 0,C 0,E1 0.1598,E2 90.0713} C_DIS
LIN {X -4.2658,Y -3.7648,Z 31,A -3.0308,B 0,C 0,E1 0.1598,E2 90.0712} C_DIS
LIN {X -3.3614,Y -4.5921,Z 31,A -3.0327,B 0,C 0,E1 0.1598,E2 90.0712} C_DIS
LIN {X -2.5113,Y -5.1016,Z 31,A -3.0233,B 0,C 0,E1 0.1598,E2 90.0714} C_DIS
LIN {X -1.7773,Y -5.4012,Z 31,A -3.0092,B 0,C 0,E1 0.1598,E2 90.0715} C_DIS
LIN {X -1.0087,Y -5.5956,Z 31,A -2.9892,B 0,C 0,E1 0.1598,E2 90.0715} C_DIS
LIN {X -0.0222,Y -5.6862,Z 31,A -2.9569,B 0,C 0,E1 0.1598,E2 90.0716} C_DIS
Enddeposition()
LIN {X -0.0222,Y -5.6862,Z 31,A -2.9569,B 0,C 0,E1 0.1598,E2 90.0716} C_DIS
Startdeposition()
$VEL.CP = VEL_PRINT
LIN {X -0.6095,Y -6.5919,Z 31,A -3.0165,B 0,C 0,E1 0.1598,E2 90.071} C_DIS
LIN {X -1.3404,Y -6.4847,Z 31,A -3.0393,B 0,C 0,E1 0.1598,E2 90.0715} C_DIS
LIN {X -2.0539,Y -6.2932,Z 31,A -3.0574,B 0,C 0,E1 0.1598,E2 90.0715} C_DIS
LIN {X -2.7422,Y -6.0247,Z 31,A -3.0712,B 0,C 0,E1 0.1598,E2 90.0715} C_DIS
LIN {X -3.3967,Y -5.6822,Z 31,A -3.0807,B 0,C 0,E1 0.1598,E2 90.0714} C_DIS
LIN {X -4.0095,Y -5.2697,Z 31,A -3.0856,B 0,C 0,E1 0.1598,E2 90.0714} C_DIS
LIN {X -4.5698,Y -4.7883,Z 31,A -3.0858,B 0,C 0,E1 0.1598,E2 90.0714} C_DIS
LIN {X -5.0747,Y -4.2492,Z 31,A -3.0814,B 0,C 0,E1 0.1598,E2 90.0714} C_DIS
LIN {X -5.5163,Y -3.6571,Z 31,A -3.0726,B 0,C 0,E1 0.1598,E2 90.0713} C_DIS
LIN {X -5.8904,Y -3.0201,Z 31,A -3.0593,B 0,C 0,E1 0.1598,E2 90.0713} C_DIS
LIN {X -6.1895,Y -2.3448,Z 31,A -3.0417,B 0,C 0,E1 0.1598,E2 90.0713} C_DIS
LIN {X -6.4115,Y -1.6403,Z 31,A -3.0201,B 0,C 0,E1 0.1598,E2 90.0713} C_DIS
LIN {X -6.557,Y -0.9162,Z 31,A -2.9948,B 0,C 0,E1 0.1598,E2 90.0713} C_DIS
LIN {X -6.6186,Y -0.1801,Z 31,A -2.9659,B 0,C 0,E1 0.1598,E2 90.0713} C_DIS
LIN {X -6.595,Y 0.5583,Z 31,A -2.9338,B 0,C 0,E1 0.1598,E2 90.0713} C_DIS
LIN {X -6.4943,Y 1.29,Z 31,A -2.8992,B 0,C 0,E1 0.1598,E2 90.0714} C_DIS
LIN {X -6.3071,Y 2.0046,Z 31,A -2.8622,B 0,C 0,E1 0.1598,E2 90.0714} C_DIS
LIN {X -6.0452,Y 2.6952,Z 31,A -2.8234,B 0,C 0,E1 0.1598,E2 90.0716} C_DIS
LIN {X -5.7078,Y 3.3521,Z 31,A -2.7832,B 0,C 0,E1 0.1598,E2 90.0716} C_DIS
LIN {X -5.2975,Y 3.9662,Z 31,A -2.7422,B 0,C 0,E1 0.1598,E2 90.0717} C_DIS
LIN {X -4.8227,Y 4.532,Z 31,A -2.7008,B 0,C 0,E1 0.1598,E2 90.0718} C_DIS
LIN {X -4.2903,Y 5.0442,Z 31,A -2.6596,B 0,C 0,E1 0.1598,E2 90.0718} C_DIS
LIN {X -3.7009,Y 5.4895,Z 31,A -2.619,B 0,C 0,E1 0.1598,E2 90.072} C_DIS
LIN {X -3.0659,Y 5.867,Z 31,A -2.5797,B 0,C 0,E1 0.1598,E2 90.072} C_DIS
LIN {X -2.393,Y 6.1722,Z 31,A -2.542,B 0,C 0,E1 0.1598,E2 90.0721} C_DIS
LIN {X -1.6901,Y 6.3994,Z 31,A -2.5065,B 0,C 0,E1 0.1598,E2 90.0722} C_DIS
LIN {X -0.9665,Y 6.5475,Z 31,A -2.4735,B 0,C 0,E1 0.1598,E2 90.0722} C_DIS
LIN {X -0.2311,Y 6.6152,Z 31,A -2.4435,B 0,C 0,E1 0.1598,E2 90.0723} C_DIS
LIN {X 0.5074,Y 6.5989,Z 31,A -2.417,B 0,C 0,E1 0.1598,E2 90.0723} C_DIS
LIN {X 1.4216,Y 6.4691,Z 31,A -2.3887,B 0,C 0,E1 0.1598,E2 90.0723} C_DIS
LIN {X 2.4783,Y 6.138,Z 31,A -2.3637,B 0,C 0,E1 0.1598,E2 90.0723} C_DIS
LIN {X 3.1881,Y 5.7983,Z 31,A -2.3519,B 0,C 0,E1 0.1598,E2 90.0723} C_DIS
LIN {X 3.8542,Y 5.3792,Z 31,A -2.3451,B 0,C 0,E1 0.1598,E2 90.0723} C_DIS
LIN {X 4.4654,Y 4.8837,Z 31,A -2.3436,B 0,C 0,E1 0.1598,E2 90.0723} C_DIS
LIN {X 5.0137,Y 4.3192,Z 31,A -2.3473,B 0,C 0,E1 0.1598,E2 90.0723} C_DIS
LIN {X 5.4912,Y 3.6936,Z 31,A -2.3562,B 0,C 0,E1 0.1598,E2 90.0722} C_DIS
LIN {X 5.8899,Y 3.0151,Z 31,A -2.3704,B 0,C 0,E1 0.1598,E2 90.0722} C_DIS
LIN {X 6.2068,Y 2.2949,Z 31,A -2.3893,B 0,C 0,E1 0.1598,E2 90.0721} C_DIS
LIN {X 6.4355,Y 1.5419,Z 31,A -2.4129,B 0,C 0,E1 0.1598,E2 90.0721} C_DIS
LIN {X 6.5747,Y 0.7673,Z 31,A -2.4407,B 0,C 0,E1 0.1598,E2 90.072} C_DIS
LIN {X 6.6197,Y -0.0186,Z 31,A -2.4725,B 0,C 0,E1 0.1598,E2 90.072} C_DIS
LIN {X 6.5691,Y -0.804,Z 31,A -2.5078,B 0,C 0,E1 0.1598,E2 90.0719} C_DIS
LIN {X 6.427,Y -1.5779,Z 31,A -2.546,B 0,C 0,E1 0.1598,E2 90.0719} C_DIS
LIN {X 6.1943,Y -2.3297,Z 31,A -2.5866,B 0,C 0,E1 0.1598,E2 90.0719} C_DIS
LIN {X 5.8752,Y -3.0492,Z 31,A -2.629,B 0,C 0,E1 0.1598,E2 90.0718} C_DIS
LIN {X 5.4706,Y -3.7243,Z 31,A -2.6726,B 0,C 0,E1 0.1598,E2 90.0718} C_DIS
LIN {X 4.992,Y -4.3492,Z 31,A -2.7168,B 0,C 0,E1 0.1598,E2 90.0718} C_DIS
LIN {X 4.44,Y -4.9102,Z 31,A -2.761,B 0,C 0,E1 0.1598,E2 90.0718} C_DIS
LIN {X 3.8256,Y -5.402,Z 31,A -2.8045,B 0,C 0,E1 0.1598,E2 90.0718} C_DIS
LIN {X 3.1567,Y -5.817,Z 31,A -2.8468,B 0,C 0,E1 0.1598,E2 90.0717} C_DIS
LIN {X 2.4438,Y -6.1505,Z 31,A -2.8871,B 0,C 0,E1 0.1598,E2 90.0717} C_DIS
LIN {X 1.6966,Y -6.3971,Z 31,A -2.925,B 0,C 0,E1 0.1598,E2 90.0717} C_DIS
LIN {X 0.9251,Y -6.5526,Z 31,A -2.96,B 0,C 0,E1 0.1598,E2 90.0717} C_DIS
LIN {X -0.056,Y -6.623,Z 31,A -2.999,B 0,C 0,E1 0.1598,E2 90.0716} C_DIS
Enddeposition()
LIN {X -0.056,Y -6.623,Z 31,A -2.999,B 0,C 0,E1 0.1598,E2 90.0716} C_DIS
Startdeposition()
$VEL.CP = VEL_PRINT
LIN {X 0.2933,Y -7.5523,Z 31,A -3.0252,B 0,C 0,E1 0.1598,E2 90.071} C_DIS
LIN {X 1.4008,Y -7.4225,Z 31,A -2.9796,B 0,C 0,E1 0.1598,E2 90.0716} C_DIS
LIN {X 2.3668,Y -7.1774,Z 31,A -2.9338,B 0,C 0,E1 0.1598,E2 90.0716} C_DIS
LIN {X 3.3151,Y -6.7905,Z 31,A -2.8825,B 0,C 0,E1 0.1598,E2 90.0716} C_DIS
LIN {X 4.3011,Y -6.2129,Z 31,A -2.8217,B 0,C 0,E1 0.1598,E2 90.0716} C_DIS
LIN {X 5.2665,Y -5.4193,Z 31,A -2.7523,B 0,C 0,E1 0.1598,E2 90.0716} C_DIS
LIN {X 5.8954,Y -4.7228,Z 31,A -2.6996,B 0,C 0,E1 0.1598,E2 90.0717} C_DIS
LIN {X 6.3348,Y -4.114,Z 31,A -2.6576,B 0,C 0,E1 0.1598,E2 90.0718} C_DIS
LIN {X 6.7987,Y -3.2982,Z 31,A -2.6056,B 0,C 0,E1 0.1598,E2 90.0717} C_DIS
LIN {X 7.1419,Y -2.4719,Z 31,A -2.5578,B 0,C 0,E1 0.1598,E2 90.0718} C_DIS
LIN {X 7.4404,Y -1.3039,Z 31,A -2.4967,B 0,C 0,E1 0.1598,E2 90.0715} C_DIS
LIN {X 7.5344,Y -0.5889,Z 31,A -2.4631,B 0,C 0,E1 0.1598,E2 90.0719} C_DIS
LIN {X 7.548,Y 0.3867,Z 31,A -2.4209,B 0,C 0,E1 0.1598,E2 90.0718} C_DIS
LIN {X 7.4383,Y 1.3405,Z 31,A -2.3844,B 0,C 0,E1 0.1598,E2 90.0719} C_DIS
LIN {X 7.1525,Y 2.4273,Z 31,A -2.3484,B 0,C 0,E1 0.1598,E2 90.0717} C_DIS
LIN {X 6.8544,Y 3.1733,Z 31,A -2.328,B 0,C 0,E1 0.1598,E2 90.0721} C_DIS
LIN {X 6.4778,Y 3.8829,Z 31,A -2.3117,B 0,C 0,E1 0.1598,E2 90.0721} C_DIS
LIN {X 6.028,Y 4.5484,Z 31,A -2.3,B 0,C 0,E1 0.1598,E2 90.0722} C_DIS
LIN {X 5.5113,Y 5.1634,Z 31,A -2.293,B 0,C 0,E1 0.1598,E2 90.0722} C_DIS
LIN {X 4.9331,Y 5.7211,Z 31,A -2.2907,B 0,C 0,E1 0.1598,E2 90.0723} C_DIS
LIN {X 4.1332,Y 6.3284,Z 31,A -2.2943,B 0,C 0,E1 0.1598,E2 90.0723} C_DIS
LIN {X 3.2758,Y 6.8096,Z 31,A -2.3056,B 0,C 0,E1 0.1598,E2 90.0723} C_DIS
LIN {X 2.4857,Y 7.1372,Z 31,A -2.321,B 0,C 0,E1 0.1598,E2 90.0724} C_DIS
LIN {X 1.3458,Y 7.4329,Z 31,A -2.3505,B 0,C 0,E1 0.1598,E2 90.0724} C_DIS
LIN {X 0.6056,Y 7.5332,Z 31,A -2.3736,B 0,C 0,E1 0.1598,E2 90.0724} C_DIS
LIN {X -0.3771,Y 7.5486,Z 31,A -2.4093,B 0,C 0,E1 0.1598,E2 90.0724} C_DIS
LIN {X -1.4607,Y 7.4148,Z 31,A -2.4549,B 0,C 0,E1 0.1598,E2 90.0723} C_DIS
LIN {X -2.4669,Y 7.1388,Z 31,A -2.5037,B 0,C 0,E1 0.1598,E2 90.0723} C_DIS
LIN {X -3.5431,Y 6.6752,Z 31,A -2.563,B 0,C 0,E1 0.1598,E2 90.0721} C_DIS
LIN {X -4.3575,Y 6.1709,Z 31,A -2.6143,B 0,C 0,E1 0.1598,E2 90.072} C_DIS
LIN {X -4.9607,Y 5.6981,Z 31,A -2.6565,B 0,C 0,E1 0.1598,E2 90.072} C_DIS
LIN {X -5.5112,Y 5.165,Z 31,A -2.6993,B 0,C 0,E1 0.1598,E2 90.0718} C_DIS
LIN {X -6.1243,Y 4.4288,Z 31,A -2.7528,B 0,C 0,E1 0.1598,E2 90.0716} C_DIS
LIN {X -6.7771,Y 3.3344,Z 31,A -2.8227,B 0,C 0,E1 0.1598,E2 90.0712} C_DIS
LIN {X -7.2248,Y 2.2151,Z 31,A -2.8865,B 0,C 0,E1 0.1598,E2 90.0712} C_DIS
LIN {X -7.4963,Y 0.9605,Z 31,A -2.9493,B 0,C 0,E1 0.1598,E2 90.0708} C_DIS
LIN {X -7.5521,Y -0.1218,Z 31,A -2.9973,B 0,C 0,E1 0.1598,E2 90.071} C_DIS
LIN {X -7.4881,Y -0.9865,Z 31,A -3.0316,B 0,C 0,E1 0.1598,E2 90.0711} C_DIS
LIN {X -7.2525,Y -2.1266,Z 31,A -3.0709,B 0,C 0,E1 0.1598,E2 90.0709} C_DIS
LIN {X -6.8515,Y -3.1803,Z 31,A -3.1007,B 0,C 0,E1 0.1598,E2 90.0709} C_DIS
LIN {X -6.4847,Y -3.8729,Z 31,A -3.1168,B 0,C 0,E1 0.1598,E2 90.0711} C_DIS
LIN {X -6.0486,Y -4.5241,Z 31,A -3.1284,B 0,C 0,E1 0.1598,E2 90.0711} C_DIS
LIN {X -5.5473,Y -5.1266,Z 31,A -3.1356,B 0,C 0,E1 0.1598,E2 90.0711} C_DIS
LIN {X -4.9862,Y -5.6739,Z 31,A -3.1382,B 0,C 0,E1 0.1598,E2 90.0712} C_DIS
LIN {X -4.0548,Y -6.3771,Z 31,A -3.1337,B 0,C 0,E1 0.1598,E2 90.0712} C_DIS
LIN {X -3.1372,Y -6.8707,Z 31,A -3.1211,B 0,C 0,E1 0.1598,E2 90.0712} C_DIS
LIN {X -2.1635,Y -7.241,Z 31,A -3.1011,B 0,C 0,E1 0.1598,E2 90.0713} C_DIS
LIN {X -1.0029,Y -7.4863,Z 31,A -3.0691,B 0,C 0,E1 0.1598,E2 90.0714} C_DIS
LIN {X -0.2455,Y -7.5534,Z 31,A -3.0442,B 0,C 0,E1 0.1598,E2 90.0715} C_DIS
LIN {X -0.2455,Y -7.5534,Z 31,A -3.0442,B 0,C 0,E1 0.1598,E2 90.0715} C_DIS
Enddeposition()
LIN {X -0.0778,Y -8.4901,Z 31,A -3.0769,B 0,C 0,E1 0.1598,E2 90.0703} C_DIS
Startdeposition()
$VEL.CP = VEL_PRINT
LIN {X -1.0305,Y -8.4256,Z 31,A -3.1101,B 0,C 0,E1 0.1598,E2 90.0714} C_DIS
LIN {X -2.0965,Y -8.2275,Z 31,A -3.1408,B 0,C 0,E1 0.1598,E2 90.0714} C_DIS
LIN {X -3.0953,Y -7.9028,Z 31,A -3.1636,B 0,C 0,E1 0.1598,E2 90.0713} C_DIS
LIN {X -3.8614,Y -7.5575,Z 31,A -3.1771,B 0,C 0,E1 0.1598,E2 90.0713} C_DIS
LIN {X -4.5896,Y -7.1384,Z 31,A -3.186,B 0,C 0,E1 0.1598,E2 90.0713} C_DIS
LIN {X -5.2729,Y -6.6495,Z 31,A -3.1903,B 0,C 0,E1 0.1598,E2 90.0712} C_DIS
LIN {X -5.9046,Y -6.0955,Z 31,A -3.1899,B 0,C 0,E1 0.1598,E2 90.0712} C_DIS
LIN {X -6.4785,Y -5.4819,Z 31,A -3.185,B 0,C 0,E1 0.1598,E2 90.0712} C_DIS
LIN {X -6.989,Y -4.8146,Z 31,A -3.1755,B 0,C 0,E1 0.1598,E2 90.0711} C_DIS
LIN {X -7.4309,Y -4.1001,Z 31,A -3.1614,B 0,C 0,E1 0.1598,E2 90.0711} C_DIS
LIN {X -7.7999,Y -3.3453,Z 31,A -3.143,B 0,C 0,E1 0.1598,E2 90.0711} C_DIS
LIN {X -8.0922,Y -2.5577,Z 31,A -3.1205,B 0,C 0,E1 0.1598,E2 90.0711} C_DIS
LIN {X -8.3693,Y -1.4311,Z 31,A -3.0828,B 0,C 0,E1 0.1598,E2 90.0708} C_DIS
LIN {X -8.4808,Y -0.4303,Z 31,A -3.0446,B 0,C 0,E1 0.1598,E2 90.0709} C_DIS
LIN {X -8.4717,Y 0.5656,Z 31,A -3.0023,B 0,C 0,E1 0.1598,E2 90.071} C_DIS
LIN {X -8.2929,Y 1.8105,Z 31,A -2.9429,B 0,C 0,E1 0.1598,E2 90.0708} C_DIS
LIN {X -7.9676,Y 2.9328,Z 31,A -2.8837,B 0,C 0,E1 0.1598,E2 90.0711} C_DIS
LIN {X -7.5382,Y 3.9003,Z 31,A -2.8273,B 0,C 0,E1 0.1598,E2 90.0714} C_DIS
LIN {X -7.1114,Y 4.6317,Z 31,A -2.7808,B 0,C 0,E1 0.1598,E2 90.0716} C_DIS
LIN {X -6.6149,Y 5.3177,Z 31,A -2.7336,B 0,C 0,E1 0.1598,E2 90.0716} C_DIS
LIN {X -6.0521,Y 5.9506,Z 31,A -2.6862,B 0,C 0,E1 0.1598,E2 90.0718} C_DIS
LIN {X -5.4292,Y 6.5243,Z 31,A -2.639,B 0,C 0,E1 0.1598,E2 90.0718} C_DIS
LIN {X -4.7523,Y 7.0332,Z 31,A -2.5926,B 0,C 0,E1 0.1598,E2 90.072} C_DIS
LIN {X -4.0281,Y 7.472,Z 31,A -2.5474,B 0,C 0,E1 0.1598,E2 90.072} C_DIS
LIN {X -3.2636,Y 7.8364,Z 31,A -2.5038,B 0,C 0,E1 0.1598,E2 90.0722} C_DIS
LIN {X -2.4665,Y 8.1222,Z 31,A -2.4623,B 0,C 0,E1 0.1598,E2 90.0722} C_DIS
LIN {X -1.6448,Y 8.3274,Z 31,A -2.4233,B 0,C 0,E1 0.1598,E2 90.0723} C_DIS
LIN {X -0.5959,Y 8.4696,Z 31,A -2.3786,B 0,C 0,E1 0.1598,E2 90.0723} C_DIS
LIN {X 0.766,Y 8.4576,Z 31,A -2.3288,B 0,C 0,E1 0.1598,E2 90.0725} C_DIS
LIN {X 1.8976,Y 8.2729,Z 31,A -2.2948,B 0,C 0,E1 0.1598,E2 90.0725} C_DIS
LIN {X 2.7144,Y 8.0418,Z 31,A -2.2744,B 0,C 0,E1 0.1598,E2 90.0725} C_DIS
LIN {X 3.5041,Y 7.7304,Z 31,A -2.2584,B 0,C 0,E1 0.1598,E2 90.0725} C_DIS
LIN {X 4.2588,Y 7.3416,Z 31,A -2.247,B 0,C 0,E1 0.1598,E2 90.0725} C_DIS
LIN {X 4.9709,Y 6.8795,Z 31,A -2.2403,B 0,C 0,E1 0.1598,E2 90.0725} C_DIS
LIN {X 5.6333,Y 6.3486,Z 31,A -2.2384,B 0,C 0,E1 0.1598,E2 90.0725} C_DIS
LIN {X 6.2395,Y 5.7543,Z 31,A -2.2413,B 0,C 0,E1 0.1598,E2 90.0724} C_DIS
LIN {X 6.7834,Y 5.1025,Z 31,A -2.2489,B 0,C 0,E1 0.1598,E2 90.0724} C_DIS
LIN {X 7.2594,Y 4.3997,Z 31,A -2.2612,B 0,C 0,E1 0.1598,E2 90.0723} C_DIS
LIN {X 7.7542,Y 3.461,Z 31,A -2.2826,B 0,C 0,E1 0.1598,E2 90.0719} C_DIS
LIN {X 8.1383,Y 2.4219,Z 31,A -2.3126,B 0,C 0,E1 0.1598,E2 90.0719} C_DIS
LIN {X 8.4022,Y 1.1965,Z 31,A -2.3548,B 0,C 0,E1 0.1598,E2 90.0715} C_DIS
LIN {X 8.4905,Y 0.0976,Z 31,A -2.3985,B 0,C 0,E1 0.1598,E2 90.0715} C_DIS
LIN {X 8.4114,Y -1.1296,Z 31,A -2.4536,B 0,C 0,E1 0.1598,E2 90.0714} C_DIS
LIN {X 8.2821,Y -1.8736,Z 31,A -2.4905,B 0,C 0,E1 0.1598,E2 90.0718} C_DIS
LIN {X 7.9408,Y -3.0056,Z 31,A -2.551,B 0,C 0,E1 0.1598,E2 90.0714} C_DIS
LIN {X 7.4976,Y -3.9758,Z 31,A -2.6089,B 0,C 0,E1 0.1598,E2 90.0716} C_DIS
LIN {X 6.8707,Y -4.991,Z 31,A -2.6752,B 0,C 0,E1 0.1598,E2 90.0715} C_DIS
LIN {X 6.1903,Y -5.8047,Z 31,A -2.735,B 0,C 0,E1 0.1598,E2 90.0716} C_DIS
LIN {X 5.4213,Y -6.535,Z 31,A -2.7943,B 0,C 0,E1 0.1598,E2 90.0716} C_DIS
LIN {X 4.3971,Y -7.261,Z 31,A -2.8629,B 0,C 0,E1 0.1598,E2 90.0716} C_DIS
LIN {X 3.65,Y -7.664,Z 31,A -2.9076,B 0,C 0,E1 0.1598,E2 90.0716} C_DIS
LIN {X 2.8662,Y -7.9902,Z 31,A -2.9502,B 0,C 0,E1 0.1598,E2 90.0716} C_DIS
LIN {X 2.0538,Y -8.2363,Z 31,A -2.9905,B 0,C 0,E1 0.1598,E2 90.0716} C_DIS
LIN {X 1.2208,Y -8.3998,Z 31,A -3.028,B 0,C 0,E1 0.1598,E2 90.0716} C_DIS
LIN {X -0.0778,Y -8.4901,Z 31,A -3.0794,B 0,C 0,E1 0.1598,E2 90.0715} C_DIS
Enddeposition()
LIN {X 0.0007,Y -4.753,Z 32,A -2.9029,B 0,C 0,E1 0.1598,E2 90.0604} C_DIS
Startdeposition()
$VEL.CP = VEL_PRINT
LIN {X 0.0007,Y -4.753,Z 32,A -2.9086,B 0,C 0,E1 0.1598,E2 90.0661} C_DIS
LIN {X 0.8351,Y -4.6788,Z 32,A -2.8797,B 0,C 0,E1 0.1598,E2 90.0711} C_DIS
LIN {X 1.4851,Y -4.5147,Z 32,A -2.8495,B 0,C 0,E1 0.1598,E2 90.0717} C_DIS
LIN {X 2.1055,Y -4.2605,Z 32,A -2.8159,B 0,C 0,E1 0.1598,E2 90.0717} C_DIS
LIN {X 2.683,Y -3.9201,Z 32,A -2.7802,B 0,C 0,E1 0.1598,E2 90.0718} C_DIS
LIN {X 3.3285,Y -3.3869,Z 32,A -2.7338,B 0,C 0,E1 0.1598,E2 90.0718} C_DIS
LIN {X 3.8728,Y -2.7508,Z 32,A -2.6866,B 0,C 0,E1 0.1598,E2 90.0718} C_DIS
LIN {X 4.2227,Y -2.179,Z 32,A -2.6495,B 0,C 0,E1 0.1598,E2 90.0718} C_DIS
LIN {X 4.4861,Y -1.5626,Z 32,A -2.6136,B 0,C 0,E1 0.1598,E2 90.0718} C_DIS
LIN {X 4.6616,Y -0.9158,Z 32,A -2.5796,B 0,C 0,E1 0.1598,E2 90.0719} C_DIS
LIN {X 4.7447,Y -0.2507,Z 32,A -2.5482,B 0,C 0,E1 0.1598,E2 90.0719} C_DIS
LIN {X 4.7328,Y 0.4194,Z 32,A -2.5201,B 0,C 0,E1 0.1598,E2 90.0719} C_DIS
LIN {X 4.6267,Y 1.0812,Z 32,A -2.4959,B 0,C 0,E1 0.1598,E2 90.0719} C_DIS
LIN {X 4.3634,Y 1.8761,Z 32,A -2.4716,B 0,C 0,E1 0.1598,E2 90.0719} C_DIS
LIN {X 4.0559,Y 2.4715,Z 32,A -2.4578,B 0,C 0,E1 0.1598,E2 90.0721} C_DIS
LIN {X 3.6677,Y 3.0177,Z 32,A -2.449,B 0,C 0,E1 0.1598,E2 90.0721} C_DIS
LIN {X 3.3299,Y 3.3902,Z 32,A -2.4457,B 0,C 0,E1 0.1598,E2 90.0721} C_DIS
LIN {X 2.8191,Y 3.8244,Z 32,A -2.446,B 0,C 0,E1 0.1598,E2 90.0721} C_DIS
LIN {X 2.1028,Y 4.2581,Z 32,A -2.454,B 0,C 0,E1 0.1598,E2 90.0721} C_DIS
LIN {X 1.6418,Y 4.459,Z 32,A -2.4626,B 0,C 0,E1 0.1598,E2 90.0722} C_DIS
LIN {X 0.9981,Y 4.6462,Z 32,A -2.4784,B 0,C 0,E1 0.1598,E2 90.0722} C_DIS
LIN {X 0.3344,Y 4.7392,Z 32,A -2.4989,B 0,C 0,E1 0.1598,E2 90.0722} C_DIS
LIN {X -0.336,Y 4.74,Z 32,A -2.5236,B 0,C 0,E1 0.1598,E2 90.0722} C_DIS
LIN {X -0.9994,Y 4.6444,Z 32,A -2.5521,B 0,C 0,E1 0.1598,E2 90.0722} C_DIS
LIN {X -1.643,Y 4.4574,Z 32,A -2.5837,B 0,C 0,E1 0.1598,E2 90.0722} C_DIS
LIN {X -2.2537,Y 4.1819,Z 32,A -2.6179,B 0,C 0,E1 0.1598,E2 90.072} C_DIS
LIN {X -2.8197,Y 3.8229,Z 32,A -2.6539,B 0,C 0,E1 0.1598,E2 90.072} C_DIS
LIN {X -3.3302,Y 3.3886,Z 32,A -2.6911,B 0,C 0,E1 0.1598,E2 90.0719} C_DIS
LIN {X -3.7734,Y 2.8857,Z 32,A -2.7286,B 0,C 0,E1 0.1598,E2 90.0719} C_DIS
LIN {X -4.1421,Y 2.326,Z 32,A -2.7658,B 0,C 0,E1 0.1598,E2 90.0717} C_DIS
LIN {X -4.4292,Y 1.7203,Z 32,A -2.802,B 0,C 0,E1 0.1598,E2 90.0717} C_DIS
LIN {X -4.6275,Y 1.08,Z 32,A -2.8364,B 0,C 0,E1 0.1598,E2 90.0716} C_DIS
LIN {X -4.7341,Y 0.4181,Z 32,A -2.8683,B 0,C 0,E1 0.1598,E2 90.0716} C_DIS
LIN {X -4.7456,Y -0.2522,Z 32,A -2.897,B 0,C 0,E1 0.1598,E2 90.0715} C_DIS
LIN {X -4.6624,Y -0.9174,Z 32,A -2.9221,B 0,C 0,E1 0.1598,E2 90.0715} C_DIS
LIN {X -4.487,Y -1.5643,Z 32,A -2.9431,B 0,C 0,E1 0.1598,E2 90.0715} C_DIS
LIN {X -4.2216,Y -2.1797,Z 32,A -2.9594,B 0,C 0,E1 0.1598,E2 90.0715} C_DIS
LIN {X -3.8724,Y -2.7518,Z 32,A -2.9708,B 0,C 0,E1 0.1598,E2 90.0715} C_DIS
LIN {X -3.4469,Y -3.2697,Z 32,A -2.9771,B 0,C 0,E1 0.1598,E2 90.0715} C_DIS
LIN {X -2.9516,Y -3.7213,Z 32,A -2.9781,B 0,C 0,E1 0.1598,E2 90.0715} C_DIS
LIN {X -2.3984,Y -4.0997,Z 32,A -2.9739,B 0,C 0,E1 0.1598,E2 90.0715} C_DIS
LIN {X -1.7977,Y -4.3967,Z 32,A -2.9645,B 0,C 0,E1 0.1598,E2 90.0715} C_DIS
LIN {X -1.1612,Y -4.6063,Z 32,A -2.95,B 0,C 0,E1 0.1598,E2 90.0716} C_DIS
LIN {X -0.5015,Y -4.7252,Z 32,A -2.9309,B 0,C 0,E1 0.1598,E2 90.0716} C_DIS
LIN {X -0.5015,Y -4.7252,Z 32,A -2.9309,B 0,C 0,E1 0.1598,E2 90.0716} C_DIS
Enddeposition()
LIN {X 0.0128,Y -5.6859,Z 32,A -2.9517,B 0,C 0,E1 0.1598,E2 90.0704} C_DIS
Startdeposition()
$VEL.CP = VEL_PRINT
LIN {X -0.8985,Y -5.6136,Z 32,A -2.9832,B 0,C 0,E1 0.1598,E2 90.0715} C_DIS
LIN {X -1.6117,Y -5.4515,Z 32,A -3.0026,B 0,C 0,E1 0.1598,E2 90.0715} C_DIS
LIN {X -2.2984,Y -5.1991,Z 32,A -3.017,B 0,C 0,E1 0.1598,E2 90.0715} C_DIS
LIN {X -2.9468,Y -4.8608,Z 32,A -3.0264,B 0,C 0,E1 0.1598,E2 90.0715} C_DIS
LIN {X -3.547,Y -4.4426,Z 32,A -3.0307,B 0,C 0,E1 0.1598,E2 90.0715} C_DIS
LIN {X -4.3348,Y -3.6846,Z 32,A -3.0273,B 0,C 0,E1 0.1598,E2 90.0712} C_DIS
LIN {X -5.0783,Y -2.5561,Z 32,A -3.0065,B 0,C 0,E1 0.1598,E2 90.0709} C_DIS
LIN {X -5.392,Y -1.8007,Z 32,A -2.9864,B 0,C 0,E1 0.1598,E2 90.0713} C_DIS
LIN {X -5.5951,Y -1.0085,Z 32,A -2.9603,B 0,C 0,E1 0.1598,E2 90.0713} C_DIS
LIN {X -5.6824,Y -0.1951,Z 32,A -2.9291,B 0,C 0,E1 0.1598,E2 90.0713} C_DIS
LIN {X -5.6504,Y 0.6222,Z 32,A -2.8934,B 0,C 0,E1 0.1598,E2 90.0713} C_DIS
LIN {X -5.5027,Y 1.4266,Z 32,A -2.8539,B 0,C 0,E1 0.1598,E2 90.0714} C_DIS
LIN {X -5.2406,Y 2.2013,Z 32,A -2.8116,B 0,C 0,E1 0.1598,E2 90.0715} C_DIS
LIN {X -4.8682,Y 2.9293,Z 32,A -2.7671,B 0,C 0,E1 0.1598,E2 90.0716} C_DIS
LIN {X -4.3984,Y 3.5984,Z 32,A -2.7215,B 0,C 0,E1 0.1598,E2 90.0717} C_DIS
LIN {X -3.8356,Y 4.1914,Z 32,A -2.6758,B 0,C 0,E1 0.1598,E2 90.0718} C_DIS
LIN {X -3.1949,Y 4.6993,Z 32,A -2.6307,B 0,C 0,E1 0.1598,E2 90.0719} C_DIS
LIN {X -2.4874,Y 5.1091,Z 32,A -2.5874,B 0,C 0,E1 0.1598,E2 90.072} C_DIS
LIN {X -1.7285,Y 5.4129,Z 32,A -2.5466,B 0,C 0,E1 0.1598,E2 90.0721} C_DIS
LIN {X -0.9341,Y 5.6071,Z 32,A -2.5091,B 0,C 0,E1 0.1598,E2 90.0722} C_DIS
LIN {X -0.1198,Y 5.6846,Z 32,A -2.4758,B 0,C 0,E1 0.1598,E2 90.0722} C_DIS
LIN {X 0.697,Y 5.6426,Z 32,A -2.4474,B 0,C 0,E1 0.1598,E2 90.0723} C_DIS
LIN {X 1.4996,Y 5.4843,Z 32,A -2.4245,B 0,C 0,E1 0.1598,E2 90.0723} C_DIS
LIN {X 2.2712,Y 5.2126,Z 32,A -2.4076,B 0,C 0,E1 0.1598,E2 90.0723} C_DIS
LIN {X 2.9952,Y 4.8318,Z 32,A -2.397,B 0,C 0,E1 0.1598,E2 90.0723} C_DIS
LIN {X 3.6572,Y 4.3515,Z 32,A -2.3929,B 0,C 0,E1 0.1598,E2 90.0723} C_DIS
LIN {X 4.2436,Y 3.7813,Z 32,A -2.3955,B 0,C 0,E1 0.1598,E2 90.0722} C_DIS
LIN {X 4.742,Y 3.133,Z 32,A -2.4046,B 0,C 0,E1 0.1598,E2 90.0722} C_DIS
LIN {X 5.1421,Y 2.4199,Z 32,A -2.4201,B 0,C 0,E1 0.1598,E2 90.072} C_DIS
LIN {X 5.5351,Y 1.3213,Z 32,A -2.452,B 0,C 0,E1 0.1598,E2 90.0716} C_DIS
LIN {X 5.6653,Y 0.4862,Z 32,A -2.483,B 0,C 0,E1 0.1598,E2 90.0719} C_DIS
LIN {X 5.6744,Y -0.3489,Z 32,A -2.5182,B 0,C 0,E1 0.1598,E2 90.0719} C_DIS
LIN {X 5.5612,Y -1.1763,Z 32,A -2.5576,B 0,C 0,E1 0.1598,E2 90.0718} C_DIS
LIN {X 5.3277,Y -1.978,Z 32,A -2.6003,B 0,C 0,E1 0.1598,E2 90.0718} C_DIS
LIN {X 4.98,Y -2.737,Z 32,A -2.6454,B 0,C 0,E1 0.1598,E2 90.0718} C_DIS
LIN {X 4.5274,Y -3.4387,Z 32,A -2.692,B 0,C 0,E1 0.1598,E2 90.0718} C_DIS
LIN {X 3.9742,Y -4.0641,Z 32,A -2.739,B 0,C 0,E1 0.1598,E2 90.0718} C_DIS
LIN {X 3.3367,Y -4.6037,Z 32,A -2.7854,B 0,C 0,E1 0.1598,E2 90.0718} C_DIS
LIN {X 2.6258,Y -5.0421,Z 32,A -2.8302,B 0,C 0,E1 0.1598,E2 90.0718} C_DIS
LIN {X 1.859,Y -5.3729,Z 32,A -2.8724,B 0,C 0,E1 0.1598,E2 90.0717} C_DIS
LIN {X 1.0512,Y -5.5853,Z 32,A -2.9111,B 0,C 0,E1 0.1598,E2 90.0717} C_DIS
LIN {X 0.2217,Y -5.6782,Z 32,A -2.9455,B 0,C 0,E1 0.1598,E2 90.0717} C_DIS
LIN {X 0.2217,Y -5.6782,Z 32,A -2.9455,B 0,C 0,E1 0.1598,E2 90.0717} C_DIS
Enddeposition()
LIN {X -0.0196,Y -6.6231,Z 32,A -2.9935,B 0,C 0,E1 0.1598,E2 90.0704} C_DIS
Startdeposition()
$VEL.CP = VEL_PRINT
LIN {X 0.9225,Y -6.5535,Z 32,A -2.9571,B 0,C 0,E1 0.1598,E2 90.0716} C_DIS
LIN {X 1.6636,Y -6.4057,Z 32,A -2.9237,B 0,C 0,E1 0.1598,E2 90.0716} C_DIS
LIN {X 2.3832,Y -6.1748,Z 32,A -2.8875,B 0,C 0,E1 0.1598,E2 90.0717} C_DIS
LIN {X 3.0712,Y -5.8623,Z 32,A -2.8489,B 0,C 0,E1 0.1598,E2 90.0717} C_DIS
LIN {X 3.7205,Y -5.4754,Z 32,A -2.8086,B 0,C 0,E1 0.1598,E2 90.0717} C_DIS
LIN {X 4.3215,Y -5.0172,Z 32,A -2.767,B 0,C 0,E1 0.1598,E2 90.0717} C_DIS
LIN {X 4.8638,Y -4.4907,Z 32,A -2.7246,B 0,C 0,E1 0.1598,E2 90.0717} C_DIS
LIN {X 5.3435,Y -3.9066,Z 32,A -2.6821,B 0,C 0,E1 0.1598,E2 90.0718} C_DIS
LIN {X 5.7541,Y -3.2719,Z 32,A -2.64,B 0,C 0,E1 0.1598,E2 90.0718} C_DIS
LIN {X 6.0897,Y -2.5947,Z 32,A -2.5987,B 0,C 0,E1 0.1598,E2 90.0718} C_DIS
LIN {X 6.3436,Y -1.8829,Z 32,A -2.5591,B 0,C 0,E1 0.1598,E2 90.0718} C_DIS
LIN {X 6.518,Y -1.1476,Z 32,A -2.5213,B 0,C 0,E1 0.1598,E2 90.0719} C_DIS
LIN {X 6.6089,Y -0.3973,Z 32,A -2.486,B 0,C 0,E1 0.1598,E2 90.0719} C_DIS
LIN {X 6.6089,Y 0.3585,Z 32,A -2.4538,B 0,C 0,E1 0.1598,E2 90.0719} C_DIS
LIN {X 6.5268,Y 1.1098,Z 32,A -2.4248,B 0,C 0,E1 0.1598,E2 90.072} C_DIS
LIN {X 6.357,Y 1.8465,Z 32,A -2.3998,B 0,C 0,E1 0.1598,E2 90.072} C_DIS
LIN {X 6.1064,Y 2.5597,Z 32,A -2.3786,B 0,C 0,E1 0.1598,E2 90.0721} C_DIS
LIN {X 5.7746,Y 3.2387,Z 32,A -2.362,B 0,C 0,E1 0.1598,E2 90.0721} C_DIS
LIN {X 5.3668,Y 3.8752,Z 32,A -2.35,B 0,C 0,E1 0.1598,E2 90.0721} C_DIS
LIN {X 4.8895,Y 4.4613,Z 32,A -2.3427,B 0,C 0,E1 0.1598,E2 90.0722} C_DIS
LIN {X 4.3495,Y 4.9903,Z 32,A -2.3402,B 0,C 0,E1 0.1598,E2 90.0722} C_DIS
LIN {X 3.7511,Y 5.452,Z 32,A -2.3427,B 0,C 0,E1 0.1598,E2 90.0723} C_DIS
LIN {X 3.1063,Y 5.8462,Z 32,A -2.3498,B 0,C 0,E1 0.1598,E2 90.0723} C_DIS
LIN {X 2.419,Y 6.1609,Z 32,A -2.3618,B 0,C 0,E1 0.1598,E2 90.0723} C_DIS
LIN {X 1.7008,Y 6.396,Z 32,A -2.3783,B 0,C 0,E1 0.1598,E2 90.0723} C_DIS
LIN {X 0.9606,Y 6.5481,Z 32,A -2.3992,B 0,C 0,E1 0.1598,E2 90.0723} C_DIS
LIN {X 0.2079,Y 6.6146,Z 32,A -2.4242,B 0,C 0,E1 0.1598,E2 90.0723} C_DIS
LIN {X -0.5475,Y 6.5972,Z 32,A -2.4528,B 0,C 0,E1 0.1598,E2 90.0723} C_DIS
LIN {X -1.2959,Y 6.4908,Z 32,A -2.4849,B 0,C 0,E1 0.1598,E2 90.0723} C_DIS
LIN {X -2.0274,Y 6.3006,Z 32,A -2.5199,B 0,C 0,E1 0.1598,E2 90.0722} C_DIS
LIN {X -2.7323,Y 6.028,Z 32,A -2.5575,B 0,C 0,E1 0.1598,E2 90.0722} C_DIS
LIN {X -3.4028,Y 5.6793,Z 32,A -2.5969,B 0,C 0,E1 0.1598,E2 90.0721} C_DIS
LIN {X -4.0286,Y 5.2554,Z 32,A -2.6379,B 0,C 0,E1 0.1598,E2 90.072} C_DIS
LIN {X -4.6007,Y 4.7615,Z 32,A -2.6798,B 0,C 0,E1 0.1598,E2 90.0719} C_DIS
LIN {X -5.1128,Y 4.2056,Z 32,A -2.7221,B 0,C 0,E1 0.1598,E2 90.0718} C_DIS
LIN {X -5.5588,Y 3.5955,Z 32,A -2.7643,B 0,C 0,E1 0.1598,E2 90.0717} C_DIS
LIN {X -5.93,Y 2.9372,Z 32,A -2.8058,B 0,C 0,E1 0.1598,E2 90.0717} C_DIS
LIN {X -6.2261,Y 2.242,Z 32,A -2.846,B 0,C 0,E1 0.1598,E2 90.0715} C_DIS
LIN {X -6.4425,Y 1.518,Z 32,A -2.8845,B 0,C 0,E1 0.1598,E2 90.0715} C_DIS
LIN {X -6.575,Y 0.7738,Z 32,A -2.9209,B 0,C 0,E1 0.1598,E2 90.0714} C_DIS
LIN {X -6.62,Y 0.0194,Z 32,A -2.9544,B 0,C 0,E1 0.1598,E2 90.0714} C_DIS
LIN {X -6.5766,Y -0.7351,Z 32,A -2.9847,B 0,C 0,E1 0.1598,E2 90.0713} C_DIS
LIN {X -6.4517,Y -1.4804,Z 32,A -3.0116,B 0,C 0,E1 0.1598,E2 90.0713} C_DIS
LIN {X -6.2414,Y -2.2065,Z 32,A -3.0346,B 0,C 0,E1 0.1598,E2 90.0713} C_DIS
LIN {X -5.9483,Y -2.9032,Z 32,A -3.0533,B 0,C 0,E1 0.1598,E2 90.0713} C_DIS
LIN {X -5.5796,Y -3.5629,Z 32,A -3.0677,B 0,C 0,E1 0.1598,E2 90.0713} C_DIS
LIN {X -5.1368,Y -4.1756,Z 32,A -3.0774,B 0,C 0,E1 0.1598,E2 90.0713} C_DIS
LIN {X -4.6279,Y -4.7344,Z 32,A -3.0824,B 0,C 0,E1 0.1598,E2 90.0713} C_DIS
LIN {X -4.0589,Y -5.2319,Z 32,A -3.0826,B 0,C 0,E1 0.1598,E2 90.0713} C_DIS
LIN {X -3.4359,Y -5.66,Z 32,A -3.078,B 0,C 0,E1 0.1598,E2 90.0713} C_DIS
LIN {X -2.7679,Y -6.0135,Z 32,A -3.0685,B 0,C 0,E1 0.1598,E2 90.0714} C_DIS
LIN {X -2.0639,Y -6.2883,Z 32,A -3.0543,B 0,C 0,E1 0.1598,E2 90.0714} C_DIS
LIN {X -1.3335,Y -6.4822,Z 32,A -3.0358,B 0,C 0,E1 0.1598,E2 90.0715} C_DIS
LIN {X -0.586,Y -6.593,Z 32,A -3.0131,B 0,C 0,E1 0.1598,E2 90.0715} C_DIS
LIN {X -0.586,Y -6.593,Z 32,A -3.0131,B 0,C 0,E1 0.1598,E2 90.0715} C_DIS
Enddeposition()
LIN {X -0.0421,Y -7.5551,Z 32,A -3.033,B 0,C 0,E1 0.1598,E2 90.0704} C_DIS
Startdeposition()
$VEL.CP = VEL_PRINT
LIN {X -1.363,Y -7.4346,Z 32,A -3.0774,B 0,C 0,E1 0.1598,E2 90.0714} C_DIS
LIN {X -2.487,Y -7.1321,Z 32,A -3.1058,B 0,C 0,E1 0.1598,E2 90.0714} C_DIS
LIN {X -3.6192,Y -6.6334,Z 32,A -3.1261,B 0,C 0,E1 0.1598,E2 90.0713} C_DIS
LIN {X -4.7203,Y -5.9023,Z 32,A -3.1353,B 0,C 0,E1 0.1598,E2 90.0711} C_DIS
LIN {X -5.5112,Y -5.1626,Z 32,A -3.133,B 0,C 0,E1 0.1598,E2 90.0711} C_DIS
LIN {X -5.9884,Y -4.6014,Z 32,A -3.1269,B 0,C 0,E1 0.1598,E2 90.0712} C_DIS
LIN {X -6.4078,Y -3.9959,Z 32,A -3.1167,B 0,C 0,E1 0.1598,E2 90.0712} C_DIS
LIN {X -6.7677,Y -3.3532,Z 32,A -3.1027,B 0,C 0,E1 0.1598,E2 90.0712} C_DIS
LIN {X -7.1843,Y -2.3447,Z 32,A -3.075,B 0,C 0,E1 0.1598,E2 90.0709} C_DIS
LIN {X -7.4374,Y -1.3189,Z 32,A -3.041,B 0,C 0,E1 0.1598,E2 90.071} C_DIS
LIN {X -7.5381,Y -0.4798,Z 32,A -3.0093,B 0,C 0,E1 0.1598,E2 90.0712} C_DIS
LIN {X -7.5292,Y 0.6648,Z 32,A -2.9604,B 0,C 0,E1 0.1598,E2 90.071} C_DIS
LIN {X -7.2702,Y 2.0676,Z 32,A -2.8912,B 0,C 0,E1 0.1598,E2 90.0707} C_DIS
LIN {X -6.8534,Y 3.1759,Z 32,A -2.8294,B 0,C 0,E1 0.1598,E2 90.0711} C_DIS
LIN {X -6.2489,Y 4.249,Z 32,A -2.7619,B 0,C 0,E1 0.1598,E2 90.0713} C_DIS
LIN {X -5.4543,Y 5.2298,Z 32,A -2.6913,B 0,C 0,E1 0.1598,E2 90.0715} C_DIS
LIN {X -4.6678,Y 5.9378,Z 32,A -2.6326,B 0,C 0,E1 0.1598,E2 90.0718} C_DIS
LIN {X -3.5954,Y 6.6465,Z 32,A -2.5631,B 0,C 0,E1 0.1598,E2 90.0719} C_DIS
LIN {X -2.4727,Y 7.1372,Z 32,A -2.5011,B 0,C 0,E1 0.1598,E2 90.0721} C_DIS
LIN {X -1.3641,Y 7.4344,Z 32,A -2.4476,B 0,C 0,E1 0.1598,E2 90.0723} C_DIS
LIN {X -0.216,Y 7.5504,Z 32,A -2.4004,B 0,C 0,E1 0.1598,E2 90.0723} C_DIS
LIN {X 1.0452,Y 7.4848,Z 32,A -2.3566,B 0,C 0,E1 0.1598,E2 90.0724} C_DIS
LIN {X 2.3232,Y 7.191,Z 32,A -2.3218,B 0,C 0,E1 0.1598,E2 90.0724} C_DIS
LIN {X 3.2692,Y 6.8128,Z 32,A -2.3029,B 0,C 0,E1 0.1598,E2 90.0724} C_DIS
LIN {X 4.1429,Y 6.3148,Z 32,A -2.2918,B 0,C 0,E1 0.1598,E2 90.0724} C_DIS
LIN {X 4.7916,Y 5.8389,Z 32,A -2.2881,B 0,C 0,E1 0.1598,E2 90.0724} C_DIS
LIN {X 5.5271,Y 5.1531,Z 32,A -2.2899,B 0,C 0,E1 0.1598,E2 90.0722} C_DIS
LIN {X 6.2143,Y 4.299,Z 32,A -2.3008,B 0,C 0,E1 0.1598,E2 90.0721} C_DIS
LIN {X 6.8556,Y 3.181,Z 32,A -2.3244,B 0,C 0,E1 0.1598,E2 90.0717} C_DIS
LIN {X 7.2586,Y 2.0857,Z 32,A -2.3562,B 0,C 0,E1 0.1598,E2 90.0717} C_DIS
LIN {X 7.4754,Y 1.1097,Z 32,A -2.3898,B 0,C 0,E1 0.1598,E2 90.0717} C_DIS
LIN {X 7.5441,Y 0.4442,Z 32,A -2.416,B 0,C 0,E1 0.1598,E2 90.0721} C_DIS
LIN {X 7.5162,Y -0.7414,Z 32,A -2.467,B 0,C 0,E1 0.1598,E2 90.0715} C_DIS
LIN {X 7.3146,Y -1.8972,Z 32,A -2.5238,B 0,C 0,E1 0.1598,E2 90.0715} C_DIS
LIN {X 6.8949,Y -3.0958,Z 32,A -2.5902,B 0,C 0,E1 0.1598,E2 90.0715} C_DIS
LIN {X 6.3766,Y -4.0557,Z 32,A -2.6504,B 0,C 0,E1 0.1598,E2 90.0715} C_DIS
LIN {X 5.7597,Y -4.8914,Z 32,A -2.7088,B 0,C 0,E1 0.1598,E2 90.0716} C_DIS
LIN {X 5.0213,Y -5.6485,Z 32,A -2.7682,B 0,C 0,E1 0.1598,E2 90.0716} C_DIS
LIN {X 4.249,Y -6.2489,Z 32,A -2.8222,B 0,C 0,E1 0.1598,E2 90.0716} C_DIS
LIN {X 3.3686,Y -6.7605,Z 32,A -2.8763,B 0,C 0,E1 0.1598,E2 90.0716} C_DIS
LIN {X 2.4307,Y -7.1571,Z 32,A -2.9276,B 0,C 0,E1 0.1598,E2 90.0716} C_DIS
LIN {X 1.4975,Y -7.4071,Z 32,A -2.9725,B 0,C 0,E1 0.1598,E2 90.0716} C_DIS
LIN {X 0.4646,Y -7.5381,Z 32,A -3.016,B 0,C 0,E1 0.1598,E2 90.0716} C_DIS
LIN {X 0.4646,Y -7.5381,Z 32,A -3.016,B 0,C 0,E1 0.1598,E2 90.0716} C_DIS
Enddeposition()
LIN {X -0.0554,Y -8.4864,Z 32,A -3.0744,B 0,C 0,E1 0.1598,E2 90.0703} C_DIS
Startdeposition()
$VEL.CP = VEL_PRINT
LIN {X 0.9341,Y -8.4342,Z 32,A -3.037,B 0,C 0,E1 0.1598,E2 90.0715} C_DIS
LIN {X 1.7173,Y -8.311,Z 32,A -3.0031,B 0,C 0,E1 0.1598,E2 90.0715} C_DIS
LIN {X 2.4857,Y -8.1156,Z 32,A -2.9666,B 0,C 0,E1 0.1598,E2 90.0716} C_DIS
LIN {X 3.5401,Y -7.719,Z 32,A -2.9111,B 0,C 0,E1 0.1598,E2 90.0716} C_DIS
LIN {X 4.4632,Y -7.2187,Z 32,A -2.8559,B 0,C 0,E1 0.1598,E2 90.0716} C_DIS
LIN {X 5.1548,Y -6.7421,Z 32,A -2.8102,B 0,C 0,E1 0.1598,E2 90.0717} C_DIS
LIN {X 5.796,Y -6.1994,Z 32,A -2.7635,B 0,C 0,E1 0.1598,E2 90.0717} C_DIS
LIN {X 6.3803,Y -5.596,Z 32,A -2.7163,B 0,C 0,E1 0.1598,E2 90.0717} C_DIS
LIN {X 6.9023,Y -4.9379,Z 32,A -2.6691,B 0,C 0,E1 0.1598,E2 90.0717} C_DIS
LIN {X 7.3568,Y -4.2314,Z 32,A -2.6222,B 0,C 0,E1 0.1598,E2 90.0718} C_DIS
LIN {X 7.7393,Y -3.4835,Z 32,A -2.5762,B 0,C 0,E1 0.1598,E2 90.0718} C_DIS
LIN {X 8.046,Y -2.7014,Z 32,A -2.5316,B 0,C 0,E1 0.1598,E2 90.0718} C_DIS
LIN {X 8.321,Y -1.688,Z 32,A -2.4779,B 0,C 0,E1 0.1598,E2 90.0716} C_DIS
LIN {X 8.481,Y -0.427,Z 32,A -2.4179,B 0,C 0,E1 0.1598,E2 90.0713} C_DIS
LIN {X 8.4533,Y 0.7581,Z 32,A -2.3686,B 0,C 0,E1 0.1598,E2 90.0715} C_DIS
LIN {X 8.3339,Y 1.6053,Z 32,A -2.3373,B 0,C 0,E1 0.1598,E2 90.072} C_DIS
LIN {X 8.1306,Y 2.4364,Z 32,A -2.3094,B 0,C 0,E1 0.1598,E2 90.072} C_DIS
LIN {X 7.8443,Y 3.2426,Z 32,A -2.2856,B 0,C 0,E1 0.1598,E2 90.0721} C_DIS
LIN {X 7.4781,Y 4.0159,Z 32,A -2.2662,B 0,C 0,E1 0.1598,E2 90.0721} C_DIS
LIN {X 7.0355,Y 4.7481,Z 32,A -2.2514,B 0,C 0,E1 0.1598,E2 90.0722} C_DIS
LIN {X 6.5218,Y 5.4324,Z 32,A -2.2413,B 0,C 0,E1 0.1598,E2 90.0722} C_DIS
LIN {X 5.9414,Y 6.0612,Z 32,A -2.236,B 0,C 0,E1 0.1598,E2 90.0723} C_DIS
LIN {X 5.3007,Y 6.6283,Z 32,A -2.2356,B 0,C 0,E1 0.1598,E2 90.0723} C_DIS
LIN {X 4.6062,Y 7.1282,Z 32,A -2.24,B 0,C 0,E1 0.1598,E2 90.0724} C_DIS
LIN {X 3.865,Y 7.5557,Z 32,A -2.2493,B 0,C 0,E1 0.1598,E2 90.0724} C_DIS
LIN {X 3.0845,Y 7.9063,Z 32,A -2.2633,B 0,C 0,E1 0.1598,E2 90.0724} C_DIS
LIN {X 2.2729,Y 8.1774,Z 32,A -2.2818,B 0,C 0,E1 0.1598,E2 90.0724} C_DIS
LIN {X 1.4381,Y 8.3655,Z 32,A -2.3046,B 0,C 0,E1 0.1598,E2 90.0724} C_DIS
LIN {X 0.3752,Y 8.4839,Z 32,A -2.3389,B 0,C 0,E1 0.1598,E2 90.0724} C_DIS
LIN {X -0.8816,Y 8.4423,Z 32,A -2.3871,B 0,C 0,E1 0.1598,E2 90.0724} C_DIS
LIN {X -1.6339,Y 8.3324,Z 32,A -2.4195,B 0,C 0,E1 0.1598,E2 90.0724} C_DIS
LIN {X -2.7409,Y 8.0329,Z 32,A -2.473,B 0,C 0,E1 0.1598,E2 90.0722} C_DIS
LIN {X -3.4678,Y 7.7513,Z 32,A -2.5117,B 0,C 0,E1 0.1598,E2 90.0722} C_DIS
LIN {X -4.433,Y 7.2385,Z 32,A -2.569,B 0,C 0,E1 0.1598,E2 90.072} C_DIS
LIN {X -5.154,Y 6.7436,Z 32,A -2.6164,B 0,C 0,E1 0.1598,E2 90.072} C_DIS
LIN {X -5.8202,Y 6.1773,Z 32,A -2.6649,B 0,C 0,E1 0.1598,E2 90.0719} C_DIS
LIN {X -6.5693,Y 5.3812,Z 32,A -2.7259,B 0,C 0,E1 0.1598,E2 90.0716} C_DIS
LIN {X -7.1844,Y 4.5245,Z 32,A -2.7847,B 0,C 0,E1 0.1598,E2 90.0715} C_DIS
LIN {X -7.7028,Y 3.5616,Z 32,A -2.8444,B 0,C 0,E1 0.1598,E2 90.0714} C_DIS
LIN {X -8.0288,Y 2.7497,Z 32,A -2.8908,B 0,C 0,E1 0.1598,E2 90.0714} C_DIS
LIN {X -8.2699,Y 1.9086,Z 32,A -2.9351,B 0,C 0,E1 0.1598,E2 90.0713} C_DIS
LIN {X -8.4625,Y 0.7014,Z 32,A -2.9928,B 0,C 0,E1 0.1598,E2 90.0709} C_DIS
LIN {X -8.4755,Y -0.4309,Z 32,A -3.0411,B 0,C 0,E1 0.1598,E2 90.0709} C_DIS
LIN {X -8.3942,Y -1.253,Z 32,A -3.0731,B 0,C 0,E1 0.1598,E2 90.0711} C_DIS
LIN {X -8.2335,Y -2.0634,Z 32,A -3.1015,B 0,C 0,E1 0.1598,E2 90.0711} C_DIS
LIN {X -7.8815,Y -3.1613,Z 32,A -3.1347,B 0,C 0,E1 0.1598,E2 90.0708} C_DIS
LIN {X -7.2644,Y -4.3911,Z 32,A -3.1639,B 0,C 0,E1 0.1598,E2 90.0706} C_DIS
LIN {X -6.7893,Y -5.0944,Z 32,A -3.1766,B 0,C 0,E1 0.1598,E2 90.0711} C_DIS
LIN {X -6.2463,Y -5.7468,Z 32,A -3.1844,B 0,C 0,E1 0.1598,E2 90.0711} C_DIS
LIN {X -5.3501,Y -6.595,Z 32,A -3.1873,B 0,C 0,E1 0.1598,E2 90.071} C_DIS
LIN {X -4.3122,Y -7.3084,Z 32,A -3.1795,B 0,C 0,E1 0.1598,E2 90.071} C_DIS
LIN {X -3.5587,Y -7.7035,Z 32,A -3.1689,B 0,C 0,E1 0.1598,E2 90.0713} C_DIS
LIN {X -2.7696,Y -8.0214,Z 32,A -3.1535,B 0,C 0,E1 0.1598,E2 90.0713} C_DIS
LIN {X -1.9526,Y -8.2587,Z 32,A -3.1336,B 0,C 0,E1 0.1598,E2 90.0713} C_DIS
LIN {X -1.116,Y -8.4133,Z 32,A -3.1095,B 0,C 0,E1 0.1598,E2 90.0714} C_DIS
LIN {X -0.0554,Y -8.4864,Z 32,A -3.0738,B 0,C 0,E1 0.1598,E2 90.0714} C_DIS
Enddeposition()
LIN {X 0.0007,Y -4.7531,Z 33,A -2.8983,B 0,C 0,E1 0.1598,E2 90.0604} C_DIS
Startdeposition()
$VEL.CP = VEL_PRINT
LIN {X 0.0007,Y -4.7531,Z 33,A -2.904,B 0,C 0,E1 0.1598,E2 90.0661} C_DIS
LIN {X -0.8333,Y -4.6769,Z 33,A -2.9362,B 0,C 0,E1 0.1598,E2 90.071} C_DIS
LIN {X -1.4831,Y -4.5128,Z 33,A -2.9537,B 0,C 0,E1 0.1598,E2 90.0716} C_DIS
LIN {X -2.1038,Y -4.2598,Z 33,A -2.9658,B 0,C 0,E1 0.1598,E2 90.0716} C_DIS
LIN {X -2.8178,Y -3.8224,Z 33,A -2.9734,B 0,C 0,E1 0.1598,E2 90.0715} C_DIS
LIN {X -3.2083,Y -3.5054,Z 33,A -2.9743,B 0,C 0,E1 0.1598,E2 90.0715} C_DIS
LIN {X -3.6679,Y -3.0175,Z 33,A -2.9705,B 0,C 0,E1 0.1598,E2 90.0715} C_DIS
LIN {X -4.0569,Y -2.4718,Z 33,A -2.9616,B 0,C 0,E1 0.1598,E2 90.0715} C_DIS
LIN {X -4.3661,Y -1.8771,Z 33,A -2.9478,B 0,C 0,E1 0.1598,E2 90.0715} C_DIS
LIN {X -4.586,Y -1.2438,Z 33,A -2.929,B 0,C 0,E1 0.1598,E2 90.0715} C_DIS
LIN {X -4.7155,Y -0.5861,Z 33,A -2.9059,B 0,C 0,E1 0.1598,E2 90.0715} C_DIS
LIN {X -4.7515,Y 0.0832,Z 33,A -2.8789,B 0,C 0,E1 0.1598,E2 90.0715} C_DIS
LIN {X -4.6924,Y 0.7509,Z 33,A -2.8485,B 0,C 0,E1 0.1598,E2 90.0715} C_DIS
LIN {X -4.5397,Y 1.4037,Z 33,A -2.8153,B 0,C 0,E1 0.1598,E2 90.0715} C_DIS
LIN {X -4.297,Y 2.0287,Z 33,A -2.7799,B 0,C 0,E1 0.1598,E2 90.0717} C_DIS
LIN {X -3.9675,Y 2.6124,Z 33,A -2.7431,B 0,C 0,E1 0.1598,E2 90.0717} C_DIS
LIN {X -3.5606,Y 3.145,Z 33,A -2.7056,B 0,C 0,E1 0.1598,E2 90.0718} C_DIS
LIN {X -3.0821,Y 3.6142,Z 33,A -2.6681,B 0,C 0,E1 0.1598,E2 90.0719} C_DIS
LIN {X -2.543,Y 4.0123,Z 33,A -2.6315,B 0,C 0,E1 0.1598,E2 90.0719} C_DIS
LIN {X -1.9536,Y 4.3314,Z 33,A -2.5963,B 0,C 0,E1 0.1598,E2 90.0721} C_DIS
LIN {X -1.3243,Y 4.5624,Z 33,A -2.5633,B 0,C 0,E1 0.1598,E2 90.0721} C_DIS
LIN {X -0.6692,Y 4.7034,Z 33,A -2.5332,B 0,C 0,E1 0.1598,E2 90.0721} C_DIS
Enddeposition()
END
